(* PLC project mtcs_axes, Institute of Astronomy OntoManager 0.0.1 *)
(* stored: creationDateTime 2017-02-03T09:57:02.669561, modificationDateTime 2017-02-03T09:57:02.669561 *)

TYPE AxesIds : (AZI := 0, ABL := 1, ELE := 2, ROC := 3, RON := 4);
END_TYPE

TYPE AxesMoveUnits : (DEGREES := 0, RADIANS := 1, ARCSECONDS := 2);
END_TYPE

TYPE AxesAlphaUnits : (HOURS := 0, DEGREES := 1, RADIANS := 2);
END_TYPE

TYPE AxesDeltaUnits : (DEGREES := 0, RADIANS := 1);
END_TYPE

TYPE AxesMuUnits : (ARCSECONDS_PER_YEAR := 0, MILLIARCSECONDS_PER_YEAR := 1, DEGREES_PER_YEAR := 2, RADIANS_PER_YEAR := 3);
END_TYPE

TYPE AxesMoveVelocityUnits : (DEGREES_PER_SECOND := 0, ARCSECONDS_PER_SECOND := 1, RADIANS_PER_SECOND := 2, ARCSECONDS_PER_MINUTE := 3, ARCSECONDS_PER_HOUR := 4);
END_TYPE

TYPE AxesRotatorActivity : (NONE_ACTIVE := 0, ROC_ACTIVE := 1, RON_ACTIVE := 2);
END_TYPE

TYPE AxesParts : STRUCT
  azi : AxesAzimuthAxis;  (* The azimuth axis *)
  ele : AxesElevationAxis;  (* The elevation axis *)
  roc : AxesRotationAxis;  (* The cassegrain derotator axis *)
  ron : AxesRotationAxis;  (* The nasmyth derotator axis *)
  io : AxesIO;  (* I/O modules and drives *)
  configManager : ConfigManager;  (* The config manager (to load/save/activate configuration data) *)
  tpoint : AxesPointingModelsSetup;  (* The TPOINT models setup *)
END_STRUCT;
END_TYPE

TYPE AxesAzimuthAxisParts : STRUCT
  virtualAxis : AngularAxis;  (* The virtual AZI axis *)
  physicalAxis : AngularAxis;  (* The physical AZI axis *)
  ablAxis : AngularAxis;  (* The (anti-backlash) ABL axis *)
  lida1 : IncrementalEncoder;  (* The external (LIDA) encoder no. 1 *)
  lida2 : IncrementalEncoder;  (* The external (LIDA) encoder no. 2 *)
  lida3 : IncrementalEncoder;  (* The external (LIDA) encoder no. 3 *)
  lida4 : IncrementalEncoder;  (* The external (LIDA) encoder no. 4 *)
  absoluteEncoder : SSIEncoder;  (* The external absolute encoder *)
END_STRUCT;
END_TYPE

TYPE AxesElevationAxisParts : STRUCT
  virtualAxis : AngularAxis;  (* The virtual axis *)
  physicalAxis : AngularAxis;  (* The physical ELE axis *)
  lida1 : IncrementalEncoder;  (* The external (LIDA) encoder no. 1 *)
  lida2 : IncrementalEncoder;  (* The external (LIDA) encoder no. 2 *)
  absoluteEncoder : SSIEncoder;  (* The external absolute encoder *)
END_STRUCT;
END_TYPE

TYPE AxesRotationAxisParts : STRUCT
  virtualAxis : AngularAxis;  (* The virtual axis *)
  physicalAxis : AngularAxis;  (* The physical axis *)
END_STRUCT;
END_TYPE

TYPE AxesPointingModelSetupParts : STRUCT
  configManager : ConfigManager;  (* The config manager (to load/save/activate configuration data) *)
END_STRUCT;
END_TYPE

TYPE AxesPointingModelsSetupParts : STRUCT
  model0 : AxesPointingModelSetup;
  model1 : AxesPointingModelSetup;
  model2 : AxesPointingModelSetup;
  model3 : AxesPointingModelSetup;
  model4 : AxesPointingModelSetup;
  model5 : AxesPointingModelSetup;
  model6 : AxesPointingModelSetup;
  model7 : AxesPointingModelSetup;
  model8 : AxesPointingModelSetup;
  model9 : AxesPointingModelSetup;
END_STRUCT;
END_TYPE

TYPE AxesIOParts : STRUCT
  aziDrive : AX52XXDrive;  (* The AX5000 drive for the AZI en ROC motors *)
  ablDrive : AX52XXDrive;  (* The AX5000 drive for the ABL en RON motors *)
  eleDrive : AX52XXDrive;  (* The AX5000 drive for the ELE en FW motors *)
  TA_AZID : EtherCatDevice;  (* Telescope Axis - AZID *)
  TA_ABLD : EtherCatDevice;  (* Telescope Axis - ABLD *)
  TA_ELED : EtherCatDevice;  (* Telescope Axis - ELED *)
  TE_COU : EtherCatDevice;  (* Telescope Encoders - COU *)
  TE_EN1 : EtherCatDevice;  (* Telescope Encoders - EN1 *)
  TE_EN2 : EtherCatDevice;  (* Telescope Encoders - EN2 *)
  TE_EN3 : EtherCatDevice;  (* Telescope Encoders - EN3 *)
  TE_EN4 : EtherCatDevice;  (* Telescope Encoders - EN4 *)
  TE_EN5 : EtherCatDevice;  (* Telescope Encoders - EN5 *)
  TE_EN6 : EtherCatDevice;  (* Telescope Encoders - EN6 *)
  TE_EN7 : EtherCatDevice;  (* Telescope Encoders - EN7 *)
END_STRUCT;
END_TYPE

TYPE AxesProcesses : STRUCT
  initialize : Process;  (* Start initializing *)
  reset : Process;  (* Reset the axis (no homing) *)
  lock : Process;  (* Lock the system *)
  unlock : Process;  (* Unlock the system *)
  changeOperatingState : ChangeOperatingStateProcess;  (* Change the operating state (e.g. AUTO, MANUAL, ...) *)
  setTarget : AxesSetTargetProcess;  (* Set a new target *)
  point : AxesPointProcess;  (* Point the telescope to a new target *)
  pointRelative : AxesPointRelativeProcess;  (* Point the telescope relative to the current target *)
  stop : AxesStopProcess;  (* Stop the axes (i.e. stop pointing, tracking, moving, ...) *)
  quickStop : AxesStopProcess;  (* Quickly stop the axes (i.e. stop pointing, tracking, moving, ...) *)
  powerOn : AxesMultiPowerOnProcess;  (* Power on the axes *)
  powerOff : AxesPowerOffProcess;  (* Power off the axes *)
  doHoming : AxesDoHomingProcess;  (* Do a homing of the axes *)
  moveAbsolute : AxesMultiMoveProcess;  (* Move the axes in alt-azimuth to an absolute position *)
  moveRelative : AxesMultiMoveProcess;  (* Move the axes in alt-azimuth relative to the current position *)
  moveKnownPosition : AxesMoveKnownPositionProcess;  (* Move the axes to the given known position *)
  enablePointingModel : AxesEnablePointingModelProcess;  (* Enable a pointing model with the given name *)
  disablePointingModel : Process;  (* Disable the currently active pointing model *)
  setAlphaDeltaVelocity : AxesSetAlphaDeltaVelocityProcess;  (* Set an additional alpha/delta velocity (e.g. to track solar system objects) *)
END_STRUCT;
END_TYPE

TYPE AxesAzimuthAxisProcesses : STRUCT
  moveAbsolute : AxesMoveAbsoluteProcess;  (* Move the axis in an absolute way *)
  moveRelative : AxesMoveRelativeProcess;  (* Move the axis relative to the current position *)
  moveVelocity : AxesMoveVelocityProcess;  (* Move the axis endlessly with the given velocity *)
  reset : Process;  (* Reset the axis (no homing) *)
  moveOutOfLimitSwitch : AxesMoveOutOfLimitSwitchProcess;  (* Move out of a limit switch *)
  powerOn : AxesPowerOnProcess;  (* Power on the axis *)
  powerOff : AxesPowerOffProcess;  (* Power off the axis *)
  doHoming : AxesDoHomingProcess;  (* Do a homing of the axis *)
  stop : AxesStopProcess;  (* Stop the axis (i.e. stop pointing, tracking, moving, ...) *)
  quickStop : AxesStopProcess;  (* Quickly stop the axes (i.e. stop pointing, tracking, moving, ...) *)
  unlockBrake : AxesUnlockBrakeProcess;  (* Temporarily unlock the brake *)
  setPosition : AxesSetPositionProcess;  (* Set the axis to the given position *)
END_STRUCT;
END_TYPE

TYPE AxesElevationAxisProcesses : STRUCT
  moveAbsolute : AxesMoveAbsoluteProcess;  (* Move the axis in an absolute way *)
  moveRelative : AxesMoveRelativeProcess;  (* Move the axis relative to the current position *)
  moveVelocity : AxesMoveVelocityProcess;  (* Move the axis endlessly with the given velocity *)
  reset : Process;  (* Reset the axis (no homing) *)
  moveOutOfLimitSwitch : AxesMoveOutOfLimitSwitchProcess;  (* Move out of a limit switch *)
  powerOn : AxesPowerOnProcess;  (* Power on the axis *)
  powerOff : AxesPowerOffProcess;  (* Power off the axis *)
  doHoming : AxesDoHomingProcess;  (* Do a homing of the axis *)
  stop : AxesStopProcess;  (* Stop the axis (i.e. stop pointing, tracking, moving, ...) *)
  quickStop : AxesStopProcess;  (* Quickly stop the axes (i.e. stop pointing, tracking, moving, ...) *)
  setPosition : AxesSetPositionProcess;  (* Set the axis to the given position *)
  unlockBrake : AxesUnlockBrakeProcess;  (* Temporarily unlock the brake *)
END_STRUCT;
END_TYPE

TYPE AxesRotationAxisProcesses : STRUCT
  moveAbsolute : AxesMoveAbsoluteProcess;  (* Move the axis in an absolute way *)
  moveRelative : AxesMoveRelativeProcess;  (* Move the axis relative to the current position *)
  moveVelocity : AxesMoveVelocityProcess;  (* Move the axis endlessly with the given velocity *)
  reset : Process;  (* Reset the axis (no homing) *)
  moveOutOfLimitSwitch : AxesMoveOutOfLimitSwitchProcess;  (* Move out of a limit switch *)
  powerOn : AxesPowerOnProcess;  (* Power on the axis *)
  powerOff : AxesPowerOffProcess;  (* Power off the axis *)
  stop : AxesStopProcess;  (* Stop the axis (i.e. stop pointing, tracking, moving, ...) *)
  quickStop : AxesStopProcess;  (* Quickly stop the axes (i.e. stop pointing, tracking, moving, ...) *)
  setPosition : AxesSetPositionProcess;  (* Set the axis to the given position *)
END_STRUCT;
END_TYPE

TYPE AxesStatuses : STRUCT
  initializationStatus : InitializationStatus;
  healthStatus : HealthStatus;
  busyStatus : BusyStatus;
  operatingStatus : OperatingStatus;
  poweredStatus : PoweredStatus;
END_STRUCT;
END_TYPE

TYPE AxesTargetStatuses : STRUCT
  healthStatus : HealthStatus;
END_STRUCT;
END_TYPE

TYPE AxesFeedbackStatuses : STRUCT
  healthStatus : HealthStatus;
END_STRUCT;
END_TYPE

TYPE AxesAzimuthAxisStatuses : STRUCT
  busyStatus : BusyStatus;  (* Is the axis in a busy state? *)
  healthStatus : HealthStatus;  (* Is the axis in a healthy state? *)
  poweredStatus : PoweredStatus;  (* Is the axis powered on or off? *)
END_STRUCT;
END_TYPE

TYPE AxesElevationAxisStatuses : STRUCT
  busyStatus : BusyStatus;  (* Is the axis in a busy state? *)
  healthStatus : HealthStatus;  (* Is the axis in a healthy state? *)
  poweredStatus : PoweredStatus;  (* Is the axis powered on or off? *)
END_STRUCT;
END_TYPE

TYPE AxesRotationAxisStatuses : STRUCT
  busyStatus : BusyStatus;  (* Is the axis in a busy state? *)
  healthStatus : HealthStatus;  (* Is the axis in a healthy state? *)
  poweredStatus : PoweredStatus;  (* Is the axis powered on or off? *)
END_STRUCT;
END_TYPE

TYPE AxesPointingModelsSetupStatuses : STRUCT
  busyStatus : BusyStatus;  (* Is the pointing models setup in a busy state? *)
  healthStatus : HealthStatus;  (* Is the pointing models setup in a healthy state? *)
END_STRUCT;
END_TYPE

TYPE AxesIOStatuses : STRUCT
  healthStatus : HealthStatus;  (* Is the I/O in a healthy state? *)
END_STRUCT;
END_TYPE

TYPE AxesLocationConfig : STRUCT
  longitude : LREAL;  (* Observatory location: longitude [degrees, positive = E, negative = W] *)
  latitude : LREAL;  (* Observatory location: latitude [degrees, positive = N, negative = S] *)
  height : REAL;  (* Observatory location: height above sea-level [m] *)
  polarMotionX : REAL;  (* Earth polar motion x in degrees *)
  polarMotionY : REAL;  (* Earth polar motion y in degrees *)
  nutationDx : REAL;  (* Nutation adjustment dX in degrees *)
  nutationDy : REAL;  (* Nutation adjustment dY in degrees *)
END_STRUCT;
END_TYPE

TYPE AxesLocalConditionsConfig : STRUCT
  useTemperatureFromSensors : BOOL;  (* True if the temperature from the sensors should be used, false to use the temperature from the config *)
  configuredTemperature : REAL;  (* Local temperature in degrees, fixed by config *)
  configuredPressure : REAL;  (* Local temperature in hectoPascal = millibar, fixed by config *)
  useRelativeHumidityFromSensors : BOOL;  (* True if the temperature from the sensors should be used, false to use the temperature from the config *)
  configuredRelativeHumidity : REAL;  (* Local relative humidity as a fraction (0...1), fixed by config *)
  configuredObservingWavelength : REAL;  (* Observing wavelength in microns, fixed by config *)
  troposphericLapseRate : REAL;  (* Tropospheric lapse rate in K/m *)
END_STRUCT;
END_TYPE

TYPE AxesAzimuthConfig : STRUCT
  absoluteEncoderOffset : LREAL;  (* Offset in degrees, of the absolute encoder, w.r.t. zero *)
  absoluteEncoderInvert : BOOL;  (* TRUE to invert the counting direction of the absolute encoder *)
  lidasInvert : BOOL;  (* TRUE to invert the counting direction of the LIDAs *)
  moveOutOfLimitSwitchDistance : LREAL;  (* How many degrees should the moveOutOfLimitSwitch process try to move? *)
  positiveLimitSwitchInput : SINT;  (* Which input (0-7) represents the positive limit switch? *)
  negativeLimitSwitchInput : SINT;  (* Which input (0-7) represents the negative limit switch? *)
  minPositionLimitVirtualAxis : LREAL;  (* Limit the minimum position of the virtual axis to this value in degrees *)
  maxPositionLimitVirtualAxis : LREAL;  (* Limit the maximum position of the virtual axis to this value in degrees *)
  minPositionLimitPhysicalAxis : LREAL;  (* Limit the minimum position of the physical axis to this value in degrees *)
  maxPositionLimitPhysicalAxis : LREAL;  (* Limit the maximum position of the physical axis to this value in degrees *)
  velocityLimit : LREAL;  (* Limit the velocity of the axis to this value in degrees/sec *)
  accelerationLimit : LREAL;  (* Limit the acceleration (or deceleration) of the axis to this value in degrees/sec^2 *)
  minPositionSetpoint : LREAL;  (* The minimum position setpoint of the axis in degrees (should be a bit before the minPositionLimit) *)
  maxPositionSetpoint : LREAL;  (* The maximum position setpoint of the axis in degrees (should be a bit before the maxPositionLimit) *)
  maxVelocitySetpoint : LREAL;  (* The maximum velocity setpoint of the axis in degrees/sec *)
  maxAccelerationSetpoint : LREAL;  (* The maximum acceleration setpoint of the axis in degrees/sec^2 *)
  slipLimit : LREAL;  (* If the difference between the LIDA-encoder and motor-encoder positions is above this value in degrees, then we have detected slip *)
  ablMaxTorqueRiseSpeed : LREAL;  (* The ABL torque can rise maximum ... Nm/s on the telescope axis (always >0) *)
  ablMaxTorqueFallSpeed : LREAL;  (* The ABL torque can fall maximum ... Nm/s on the telescope axis (always >0) *)
  ablMaxTorque : LREAL;  (* The maximum ABL torque in Nm/s on the telescope axis (always >0) *)
  ablMinTorque : LREAL;  (* The minimum ABL torque in Nm/s on the telescope axis (always >0) *)
  ablZeroAccTorque : LREAL;  (* The ABL torque when the axis is not accelerating or decelerating (always >0) *)
  ablTorqueOutputOverride : LREAL;  (* Scale the ABL output torque by this fraction value (only for testing purposes, must be 1 normally!) *)
  ablPositiveTorque : BOOL;  (* True if a positive torque must be applied, false if a negative torque must be applied *)
  aziAndAblSameDirection : BOOL;  (* True if the AZI and ABL axes rotate in the same direction? *)
  homingHomePosition : LREAL;  (* The position of the homing mark (in degrees), with respect to the absolute zero *)
  homingStartAbsEncPosition : LREAL;  (* Absolute encoder position where the homing should go to first, in degrees *)
  homingGotoStartVelocity : LREAL;  (* Velocity when going to the start position, in degrees/sec *)
  homingVelocity : LREAL;  (* Velocity to search for the homing mark, in degrees/sec *)
  homingRange : LREAL;  (* Maximum distance to be covered while searching for the homing mark, in degrees *)
  quickStopDeceleration : LREAL;  (* Quick stop deceleration, in degrees/sec2 *)
  quickStopJerk : LREAL;  (* Quick stop jerk, in degrees/sec3 *)
END_STRUCT;
END_TYPE

TYPE AxesElevationConfig : STRUCT
  absoluteEncoderOffset : LREAL;  (* Offset in degrees, of the absolute encoder, w.r.t. zero *)
  absoluteEncoderInvert : BOOL;  (* TRUE to invert the counting direction *)
  lidasInvert : BOOL;  (* TRUE to invert the counting direction of the LIDAs *)
  moveOutOfLimitSwitchDistance : LREAL;  (* How many degrees should the moveOutOfLimitSwitch process try to move? *)
  positiveLimitSwitchInput : SINT;  (* Which input (0-7) represents the positive limit switch? *)
  negativeLimitSwitchInput : SINT;  (* Which input (0-7) represents the negative limit switch? *)
  minPositionLimitVirtualAxis : LREAL;  (* Limit the minimum position of the axis to this value in degrees, of the virtual axis *)
  maxPositionLimitVirtualAxis : LREAL;  (* Limit the maximum position of the axis to this value in degrees, of the virtual axis *)
  minPositionLimitPhysicalAxis : LREAL;  (* Limit the minimum position of the axis to this value in degrees, of the physical axis *)
  maxPositionLimitPhysicalAxis : LREAL;  (* Limit the maximum position of the axis to this value in degrees, of the physical axis *)
  velocityLimit : LREAL;  (* Limit the velocity of the axis to this value in degrees/sec *)
  accelerationLimit : LREAL;  (* Limit the acceleration (or deceleration) of the axis to this value in degrees/sec^2 *)
  minPositionSetpoint : LREAL;  (* The minimum position setpoint of the axis in degrees *)
  maxPositionSetpoint : LREAL;  (* The maximum position setpoint of the axis in degrees *)
  maxVelocitySetpoint : LREAL;  (* The maximum velocity setpoint of the axis in degrees/sec *)
  maxAccelerationSetpoint : LREAL;  (* The maximum acceleration setpoint of the axis in degrees/sec^2 *)
  slipLimit : LREAL;  (* If the difference between the LIDA-encoder and motor-encoder positions is above this value in degrees, then we have detected slip *)
  homingHomePosition : LREAL;  (* The position of the homing mark (in degrees), with respect to the absolute zero *)
  homingStartAbsEncPosition : LREAL;  (* Absolute encoder position where the homing should go to first, in degrees *)
  homingGotoStartVelocity : LREAL;  (* Velocity when going to the start position, in degrees/sec *)
  homingVelocity : LREAL;  (* Velocity to search for the homing mark, in degrees/sec *)
  homingRange : LREAL;  (* Maximum distance to be covered while searching for the homing mark, in degrees *)
  quickStopDeceleration : LREAL;  (* Quick stop deceleration, in degrees/sec2 *)
  quickStopJerk : LREAL;  (* Quick stop jerk, in degrees/sec3 *)
END_STRUCT;
END_TYPE

TYPE AxesRotationConfig : STRUCT
  motorEncoderOffset : LREAL;  (* Offset in degrees, of the absolute motor encoder, w.r.t. zero *)
  moveOutOfLimitSwitchDistance : LREAL;  (* How many degrees should the moveOutOfLimitSwitch process try to move? *)
  positiveLimitSwitchInput : SINT;  (* Which input (0-7) represents the positive limit switch? *)
  negativeLimitSwitchInput : SINT;  (* Which input (0-7) represents the negative limit switch? *)
  minPositionLimitVirtualAxis : LREAL;  (* Limit the minimum position of the axis to this value in degrees, of the virtual axis *)
  maxPositionLimitVirtualAxis : LREAL;  (* Limit the maximum position of the axis to this value in degrees, of the virtual axis *)
  minPositionLimitPhysicalAxis : LREAL;  (* Limit the minimum position of the axis to this value in degrees, of the physical axis *)
  maxPositionLimitPhysicalAxis : LREAL;  (* Limit the maximum position of the axis to this value in degrees, of the physical axis *)
  velocityLimit : LREAL;  (* Limit the velocity of the axis to this value in degrees/sec *)
  accelerationLimit : LREAL;  (* Limit the acceleration (or deceleration) of the axis to this value in degrees/sec^2 *)
  minPositionSetpoint : LREAL;  (* The minimum position setpoint of the axis in degrees *)
  maxPositionSetpoint : LREAL;  (* The maximum position setpoint of the axis in degrees *)
  maxVelocitySetpoint : LREAL;  (* The maximum velocity setpoint of the axis in degrees/sec *)
  maxAccelerationSetpoint : LREAL;  (* The maximum acceleration setpoint of the axis in degrees/sec^2 *)
  quickStopDeceleration : LREAL;  (* Quick stop deceleration, in degrees/sec2 *)
  quickStopJerk : LREAL;  (* Quick stop jerk, in degrees/sec3 *)
END_STRUCT;
END_TYPE

TYPE AxesKnownPositionConfig : STRUCT
  name : STRING;  (* The name of the position (e.g. 'PARK') *)
  allowObserver : BOOL;  (* Can an observer switch to this position? *)
  azi : LREAL;  (* Azimuth in degrees *)
  ele : LREAL;  (* Elevation in degrees *)
  roc : LREAL;  (* Cassegrain rotation in degrees *)
  ron : LREAL;  (* Nasmyth B rotation in degrees *)
  doAzi : BOOL;  (* Change the azimuth axis to the 'azi' position *)
  doEle : BOOL;  (* Change the elevation axis to the 'ele' position *)
  doRoc : BOOL;  (* Change the cassegrain rotation axis to the 'roc' position *)
  doRon : BOOL;  (* Change the nasmyth rotation axis to the 'ron' position *)
END_STRUCT;
END_TYPE

TYPE AxesKnownPositionsConfig : STRUCT
  position0 : AxesKnownPositionConfig;  (* Known position 0 *)
  position1 : AxesKnownPositionConfig;  (* Known position 1 *)
  position2 : AxesKnownPositionConfig;  (* Known position 2 *)
  position3 : AxesKnownPositionConfig;  (* Known position 3 *)
  position4 : AxesKnownPositionConfig;  (* Known position 4 *)
  position5 : AxesKnownPositionConfig;  (* Known position 5 *)
  position6 : AxesKnownPositionConfig;  (* Known position 6 *)
  position7 : AxesKnownPositionConfig;  (* Known position 7 *)
  position8 : AxesKnownPositionConfig;  (* Known position 8 *)
  position9 : AxesKnownPositionConfig;  (* Known position 9 *)
  position10 : AxesKnownPositionConfig;  (* Known position 10 *)
  position11 : AxesKnownPositionConfig;  (* Known position 11 *)
  position12 : AxesKnownPositionConfig;  (* Known position 12 *)
  position13 : AxesKnownPositionConfig;  (* Known position 13 *)
  position14 : AxesKnownPositionConfig;  (* Known position 14 *)
  position15 : AxesKnownPositionConfig;  (* Known position 15 *)
  position16 : AxesKnownPositionConfig;  (* Known position 16 *)
  position17 : AxesKnownPositionConfig;  (* Known position 17 *)
  position18 : AxesKnownPositionConfig;  (* Known position 18 *)
  position19 : AxesKnownPositionConfig;  (* Known position 19 *)
END_STRUCT;
END_TYPE

TYPE AxesConfig : STRUCT
  location : AxesLocationConfig;  (* Location of the observatory *)
  localConditions : AxesLocalConditionsConfig;  (* Location of the observatory *)
  knownPositions : AxesKnownPositionsConfig;  (* Known (predefined) positions (e.g. could be Park, Cover, Park winter, Mirror washing, ...) *)
  azi : AxesAzimuthConfig;  (* Azimuth axis *)
  ele : AxesElevationConfig;  (* Elevation axis *)
  roc : AxesRotationConfig;  (* Cassegrain rotation axis *)
  ron : AxesRotationConfig;  (* Nasmyth rotation axis *)
  cassegrainRotatorName : STRING;  (* Name of the Cassegrain rotator *)
  nasmythRotatorName : STRING;  (* Name of the Nasmyth rotator *)
  rocGuiAngle : LREAL;  (* Amgle to show ROC in the GUI *)
  ronGuiAngle : LREAL;  (* Amgle to show RON in the GUI *)
  knownPositionToleranceAzi : LREAL;  (* Tolerance (in degrees) to determine if the telescope is at a known position in azi direction *)
  knownPositionToleranceEle : LREAL;  (* Tolerance (in degrees) to determine if the telescope is at a known position in ele direction *)
  knownPositionToleranceRoc : LREAL;  (* Tolerance (in degrees) to determine if the telescope is at a known position in roc direction *)
  knownPositionToleranceRon : LREAL;  (* Tolerance (in degrees) to determine if the telescope is at a known position in ron direction *)
  rocPositionAngleSign : INT;  (* -1 to invert the sign of the PA for the cas derotator, 1 for positive *)
  ronPositionAngleSign : INT;  (* -1 to invert the sign of the PA for the cas derotator, 1 for positive *)
  tpointAziSign : INT;  (* -1 or 1 to invert input for TPOINT: A *)
  tpointEleSign : INT;  (* -1 or 1 to invert input for TPOINT: E *)
  tpointDeltaAziSign : INT;  (* -1 or 1 to invert input for TPOINT: DA *)
  tpointDeltaEleSign : INT;  (* -1 or 1 to invert input for TPOINT: DE *)
  tpointOldFormulas : BOOL;  (* True to use the old formulas *)
  tpointConvertRawAlphaDelta : BOOL;  (* If True, raw encoder values will be converted to feedback.alpha and feedback.delta, instead of corrected encoder values. Only use for tech stuff! *)
END_STRUCT;
END_TYPE

TYPE AxesPointingModelConfig : STRUCT
  name : STRING;  (* This name can be matched against the instrument name in the MTCS config and the focal station name in the M3 config. *)
  IE : LREAL;  (* Index error in elevation *)
  IA : LREAL;  (* Index error in azimuth *)
  CA : LREAL;  (* Nonperpendicularity of elevation and pointing axes *)
  AN : LREAL;  (* NS misalignment of azimuth axis *)
  AW : LREAL;  (* EW misalignment of azimuth axis *)
  NPAE : LREAL;  (* Nonperpendicularity of azimuth and elevation axes *)
  NRX : LREAL;  (* Horizontal displacement of Nasmyth rotation *)
  NRY : LREAL;  (* Vertical displacement of Nasmyth rotation *)
  ACES : LREAL;  (* Az centering error (sin component) *)
  ACEC : LREAL;  (* Az centering error (cos component) *)
  ECES : LREAL;  (* El centering error (sin component) *)
  ECEC : LREAL;  (* El centering error (cos component) *)
  TF : LREAL;  (* Tube flexure - sin(zeta) law *)
  TX : LREAL;  (* Tube flexure - tan(zeta) law *)
  FLOP : LREAL;  (* Constant vertical displacement *)
  POX : LREAL;  (* The x-coordinate of a pointing origin on a derotator *)
  POY : LREAL;  (* The y-coordinate of a pointing origin on a derotator *)
END_STRUCT;
END_TYPE

TYPE AxesSetTargetProcessArgs : STRUCT
  alphaUnits : AxesAlphaUnits;  (* The units in which alpha is given *)
  alpha : LREAL;  (* Right ascention, in the units of the alphaUnits argument *)
  deltaUnits : AxesDeltaUnits;  (* The units in which delta is given *)
  delta : LREAL;  (* Declination, in the units of the deltaUnits argument *)
  muUnits : AxesMuUnits;  (* The units in which muAlpha and muDelta are given *)
  muAlpha : LREAL;  (* Right ascention proper motion, the units of muUmits (do not multiply by cos(delta)!) *)
  muDelta : LREAL;  (* Declination proper motion, in radians/year *)
  parallax : LREAL;  (* Object parallax, in arcseconds *)
  radialVelocity : LREAL;  (* Object radial velocity, in km/s *)
  epoch : LREAL := 2000;  (* Epoch, e.g. 2000.0 *)
END_STRUCT;
END_TYPE

TYPE AxesPointProcessArgs : STRUCT
  alphaUnits : AxesAlphaUnits;  (* The units in which alpha is given *)
  alpha : LREAL;  (* Right ascention, in the units of the alphaUnits argument *)
  deltaUnits : AxesDeltaUnits;  (* The units in which delta is given *)
  delta : LREAL;  (* Declination, in the units of the deltaUnits argument *)
  muUnits : AxesMuUnits;  (* The units in which muAlpha and muDelta are given *)
  muAlpha : LREAL;  (* Right ascention proper motion, the units of muUmits (do not multiply by cos(delta)!) *)
  muDelta : LREAL;  (* Declination proper motion, in radians/year *)
  parallax : LREAL;  (* Object parallax, in arcseconds *)
  radialVelocity : LREAL;  (* Object radial velocity, in km/s *)
  epoch : LREAL := 2000;  (* Epoch, e.g. 2000.0 *)
  tracking : BOOL := TRUE;  (* True to start tracking the object, false to Only do a pointing *)
  rotUnits : AxesMoveUnits;  (* Units of the 'rot', 'roc' and 'ron' arguments (RADIANS, DEGREES, ARCSECONDS, ...) *)
  rotOffset : LREAL;  (* Offset to move the currently active rotator (incompatible with 'roc' and 'ron' args) *)
  rocOffset : LREAL;  (* Offset to move the cassegrain rotation axis (incompatible with 'rot' arg) *)
  ronOffset : LREAL;  (* Offset to move the nasmyth rotation axis (incompatible with 'rot' arg) *)
  doRotOffset : BOOL;  (* True to move the currently active rotator, false to leave it untouched *)
  doRocOffset : BOOL;  (* True to move the cassegrain rotation axis, false to leave it untouched *)
  doRonOffset : BOOL;  (* True to move the nasmyth rotation axis, false to leave it untouched *)
END_STRUCT;
END_TYPE

TYPE AxesPointRelativeProcessArgs : STRUCT
  alphaUnits : AxesAlphaUnits;  (* The units in which alpha is given *)
  alpha : LREAL;  (* Right ascention, in the units of the alphaUnits argument *)
  deltaUnits : AxesDeltaUnits;  (* The units in which delta is given *)
  delta : LREAL;  (* Declination, in the units of the deltaUnits argument *)
END_STRUCT;
END_TYPE

TYPE AxesMoveRelativeProcessArgs : STRUCT
  units : AxesMoveUnits;  (* Units of the 'value' argument (RADIANS, DEGREES, ARCSECONDS, ...) *)
  value : LREAL;  (* Move the axis with this value (which units depends on the 'units' argument) *)
END_STRUCT;
END_TYPE

TYPE AxesMoveAbsoluteProcessArgs : STRUCT
  units : AxesMoveUnits;  (* Units of the 'value' argument (RADIANS, DEGREES, ARCSECONDS, ...) *)
  value : LREAL;  (* Move the axis to this value (which units depends on the 'units' argument) + the optional offset *)
  offset : LREAL;  (* Optional extra offset (which will not be added to the 'startPos' *)
END_STRUCT;
END_TYPE

TYPE AxesMoveKnownPositionProcessArgs : STRUCT
  name : STRING;  (* Name of the position to move to *)
END_STRUCT;
END_TYPE

TYPE AxesMoveVelocityProcessArgs : STRUCT
  units : AxesMoveVelocityUnits;  (* Units of the 'value' argument (RADIANS_PER_SECOND, DEGREES_PER_SECOND, ...) *)
  value : LREAL;  (* Move the axis with this velocity (which units depends on the 'units' argument) *)
END_STRUCT;
END_TYPE

TYPE AxesMoveOutOfLimitSwitchProcessArgs : STRUCT
  switch : LimitSwitches;  (* Positive or negative limit switch *)
END_STRUCT;
END_TYPE

TYPE AxesMultiPowerOnProcessArgs : STRUCT
  azi : BOOL;  (* TRUE to power on AZI *)
  ele : BOOL;  (* TRUE to power on ELE *)
  roc : BOOL;  (* TRUE to power on ROC *)
  ron : BOOL;  (* TRUE to power on RON *)
  fw : BOOL;  (* TRUE to power on FW *)
END_STRUCT;
END_TYPE

TYPE AxesSetAlphaDeltaVelocityProcessArgs : STRUCT
  units : AxesMoveVelocityUnits;  (* Units of the alphaVelocity and deltaVelocity *)
  alphaVelocity : LREAL;  (* Velocity in alpha direction *)
  deltaVelocity : LREAL;  (* Velocity in delta direction *)
END_STRUCT;
END_TYPE

TYPE AxesMultiMoveProcessArgs : STRUCT
  units : AxesMoveUnits;  (* Units of the 'azi', 'ele', 'roc' and 'ron' arguments (RADIANS, DEGREES, ARCSECONDS, ...) *)
  azi : LREAL;  (* Angle to move the azimuth axis *)
  ele : LREAL;  (* Angle to move the elevation axis *)
  rot : LREAL;  (* Angle to move the currently active rotator (incompatible with 'roc' and 'ron' args) *)
  roc : LREAL;  (* Angle to move the cassegrain rotation axis (incompatible with 'rot' arg) *)
  ron : LREAL;  (* Angle to move the nasmyth rotation axis (incompatible with 'rot' arg) *)
  doAzi : BOOL;  (* True to move the azimuth axis, false to leave it untouched *)
  doEle : BOOL;  (* True to move the elevation axis, false to leave it untouched *)
  doRot : BOOL;  (* True to move the currently active rotator, false to leave it untouched *)
  doRoc : BOOL;  (* True to move the cassegrain rotation axis, false to leave it untouched *)
  doRon : BOOL;  (* True to move the nasmyth rotation axis, false to leave it untouched *)
  preferMostTravel : BOOL := FALSE;  (* Only in case of relative movement during tracking: If possible, go to the position where there is most travel (if the telescope is tracking). If false, it will go there the quickest way possible. *)
END_STRUCT;
END_TYPE

TYPE AxesEnablePointingModelProcessArgs : STRUCT
  name : STRING;  (* Name of the pointing model *)
END_STRUCT;
END_TYPE

TYPE AxesUnlockBrakeProcessArgs : STRUCT
  seconds : LREAL := 10.0;  (* Unlock the brake for this number of seconds (0 means forever) *)
END_STRUCT;
END_TYPE

TYPE AxesSetPositionProcessArgs : STRUCT
  value : LREAL;  (* New position to be taken over by the axis *)
END_STRUCT;
END_TYPE

FUNCTION_BLOCK SM_Axes
  VAR_INPUT
    {attribute 'OPC.UA.DA' := '1'}
    {attribute 'OPC.UA.DA.Access' := '1'}
    editableConfig : AxesConfig;  (* Editable configuration of the Axes subsystem *)
    {attribute 'OPC.UA.DA' := '1'}
    {attribute 'OPC.UA.DA.Access' := '1'}
    fromCppAxes AT %I* : TmcToPlcAxes;  (* Data from the C++ task *)
  END_VAR
  VAR_OUTPUT
    {attribute 'OPC.UA.DA' := '1'}
    {attribute 'OPC.UA.DA.Access' := '1'}
    actualStatus : STRING;  (* Current status description *)
    previousStatus : STRING;  (* Previous status description *)
    {attribute 'OPC.UA.DA' := '1'}
    {attribute 'OPC.UA.DA.Access' := '1'}
    isPoweredOffByPersonInDome : BOOL;  (* True if the axes are powered off due to a person entering the dome *)
    {attribute 'OPC.UA.DA' := '1'}
    {attribute 'OPC.UA.DA.Access' := '1'}
    isPointing : BOOL;  (* True if the telescope is pointing *)
    {attribute 'OPC.UA.DA' := '1'}
    {attribute 'OPC.UA.DA.Access' := '1'}
    isLimitsReached : BOOL;  (* True if a positiom limit is reached *)
    {attribute 'OPC.UA.DA' := '1'}
    {attribute 'OPC.UA.DA.Access' := '1'}
    isTracking : BOOL;  (* True if the telescope is tracking *)
    {attribute 'OPC.UA.DA' := '1'}
    {attribute 'OPC.UA.DA.Access' := '1'}
    isOffsetting : BOOL;  (* True if the telescope is offsetting (movin *)
    {attribute 'OPC.UA.DA' := '1'}
    {attribute 'OPC.UA.DA.Access' := '1'}
    isAtKnownPosition : BOOL;  (* True if the telescope is at a known position *)
    {attribute 'OPC.UA.DA' := '1'}
    {attribute 'OPC.UA.DA.Access' := '1'}
    isPointingModelActive : BOOL;  (* Is a pointing model currently active? *)
    {attribute 'OPC.UA.DA' := '1'}
    {attribute 'OPC.UA.DA.Access' := '1'}
    activeRotator : AxesRotatorActivity;  (* Which rotator is active? *)
    {attribute 'OPC.UA.DA' := '1'}
    {attribute 'OPC.UA.DA.Access' := '1'}
    actualKnownPositionName : STRING;  (* Name of the known position if isAtKnownPosition is True *)
    {attribute 'OPC.UA.DA' := '1'}
    {attribute 'OPC.UA.DA.Access' := '1'}
    config : AxesConfig;  (* Active configuration of the Axes subsystem *)
    {attribute 'OPC.UA.DA' := '1'}
    {attribute 'OPC.UA.DA.Access' := '1'}
    toCppAxes AT %Q* : TmcFromPlcAxes;  (* Data to the C++ task *)
    {attribute 'OPC.UA.DA' := '1'}
    {attribute 'OPC.UA.DA.Access' := '1'}
    activePointingModel : AxesPointingModelConfig;  (* Currently active TPoint model (if isPointingModelActive is TRUE) *)
    {attribute 'OPC.UA.DA' := '1'}
    {attribute 'OPC.UA.DA.Access' := '1'}
    activePointingModelNumber : INT;  (* Number of the currently active TPoint model (if isPointingModelActive is TRUE), -1 if no model is active *)
    {attribute 'OPC.UA.DA' := '1'}
    {attribute 'OPC.UA.DA.Access' := '1'}
    target : AxesTarget;  (* The actual target *)
    {attribute 'OPC.UA.DA' := '1'}
    {attribute 'OPC.UA.DA.Access' := '1'}
    feedback : AxesFeedback;  (* The actual feedback *)
    statuses : AxesStatuses;  (* Statuses of the state machine *)
    parts : AxesParts;  (* Parts of the state machine *)
    processes : AxesProcesses;  (* Processes of the state machine *)
  END_VAR
  VAR_IN_OUT
    {attribute 'OPC.UA.DA' := '0'}
    timing : ServicesTiming;  (* Reference to the timing service *)
    {attribute 'OPC.UA.DA' := '0'}
    motionBlocking : SafetyMotionBlocking;  (* Reference to the motion blocking safety *)
    {attribute 'OPC.UA.DA' := '0'}
    domeAccess : SafetyDomeAccess;  (* Reference to the dome access safety *)
    {attribute 'OPC.UA.DA' := '0'}
    operatorStatus : OperatorStatus;  (* Shared operator status *)
    {attribute 'OPC.UA.DA' := '0'}
    activityStatus : ActivityStatus;  (* Shared activity status *)
    {attribute 'OPC.UA.DA' := '0'}
    activeInstrument : InstrumentConfig;  (* Instrument config *if* isInstrumentActive is TRUE *)
    {attribute 'OPC.UA.DA' := '0'}
    isInstrumentActive : BOOL;  (* Is an instrument currently active (i.e. is M3 static at a known position?) *)
  END_VAR

            parts.azi(
    isEnabled := operatorStatus.tech,
    id := AxesIds.AZI,
    config := config.azi,
    aziDriveChannel := parts.io.parts.aziDrive.parts.channelA,
    ablDriveChannel := parts.io.parts.ablDrive.parts.channelA,
    aziMainDriveChannel := parts.io.parts.aziDrive.parts.channelA,
    ablMainDriveChannel := parts.io.parts.ablDrive.parts.channelA);
parts.ele(
    isEnabled := operatorStatus.tech,
    id := AxesIds.ELE,
    config := config.ele,
    driveChannel := parts.io.parts.eleDrive.parts.channelA,
    mainDriveChannel := parts.io.parts.eleDrive.parts.channelA);
parts.roc(
    isEnabled := operatorStatus.tech,
    id := AxesIds.ROC,
    config := config.roc,
    driveChannel := parts.io.parts.aziDrive.parts.channelB,
    mainDriveChannel := parts.io.parts.aziDrive.parts.channelA);
parts.ron(
    isEnabled := operatorStatus.tech,
    id := AxesIds.RON,
    config := config.ron,
    driveChannel := parts.io.parts.ablDrive.parts.channelB,
    mainDriveChannel := parts.io.parts.ablDrive.parts.channelA);
parts.io( isEnabled := operatorStatus.tech );
parts.configManager( isEnabled := operatorStatus.tech );
parts.tpoint( isEnabled := operatorStatus.tech );
statuses.initializationStatus();
statuses.healthStatus(
    isGood := feedback.statuses.healthStatus.isGood AND (target.statuses.healthStatus.isGood AND (parts.azi.statuses.healthStatus.isGood AND (parts.ele.statuses.healthStatus.isGood AND (parts.roc.statuses.healthStatus.isGood AND (parts.ron.statuses.healthStatus.isGood AND (parts.configManager.statuses.healthStatus.isGood AND (parts.tpoint.statuses.healthStatus.isGood AND (parts.io.statuses.healthStatus.isGood AND (processes.initialize.statuses.healthStatus.isGood AND (processes.reset.statuses.healthStatus.isGood AND (processes.lock.statuses.healthStatus.isGood AND (processes.unlock.statuses.healthStatus.isGood AND (processes.changeOperatingState.statuses.healthStatus.isGood AND (processes.setTarget.statuses.healthStatus.isGood AND (processes.point.statuses.healthStatus.isGood AND (processes.pointRelative.statuses.healthStatus.isGood AND (processes.stop.statuses.healthStatus.isGood AND (processes.quickStop.statuses.healthStatus.isGood AND (processes.powerOn.statuses.healthStatus.isGood AND (processes.powerOff.statuses.healthStatus.isGood AND (processes.doHoming.statuses.healthStatus.isGood AND (processes.moveAbsolute.statuses.healthStatus.isGood AND (processes.moveRelative.statuses.healthStatus.isGood AND (processes.moveKnownPosition.statuses.healthStatus.isGood AND (processes.enablePointingModel.statuses.healthStatus.isGood AND (processes.disablePointingModel.statuses.healthStatus.isGood AND processes.setAlphaDeltaVelocity.statuses.healthStatus.isGood)))))))))))))))))))))))))),
    hasWarning := feedback.statuses.healthStatus.hasWarning OR (target.statuses.healthStatus.hasWarning OR (parts.azi.statuses.healthStatus.hasWarning OR (parts.ele.statuses.healthStatus.hasWarning OR (parts.roc.statuses.healthStatus.hasWarning OR (parts.ron.statuses.healthStatus.hasWarning OR (parts.configManager.statuses.healthStatus.hasWarning OR (parts.tpoint.statuses.healthStatus.hasWarning OR (parts.io.statuses.healthStatus.hasWarning OR (processes.initialize.statuses.healthStatus.hasWarning OR (processes.reset.statuses.healthStatus.hasWarning OR (processes.lock.statuses.healthStatus.hasWarning OR (processes.unlock.statuses.healthStatus.hasWarning OR (processes.changeOperatingState.statuses.healthStatus.hasWarning OR (processes.setTarget.statuses.healthStatus.hasWarning OR (processes.point.statuses.healthStatus.hasWarning OR (processes.pointRelative.statuses.healthStatus.hasWarning OR (processes.stop.statuses.healthStatus.hasWarning OR (processes.quickStop.statuses.healthStatus.hasWarning OR (processes.powerOn.statuses.healthStatus.hasWarning OR (processes.powerOff.statuses.healthStatus.hasWarning OR (processes.doHoming.statuses.healthStatus.hasWarning OR (processes.moveAbsolute.statuses.healthStatus.hasWarning OR (processes.moveRelative.statuses.healthStatus.hasWarning OR (processes.moveKnownPosition.statuses.healthStatus.hasWarning OR (processes.enablePointingModel.statuses.healthStatus.hasWarning OR (processes.disablePointingModel.statuses.healthStatus.hasWarning OR processes.setAlphaDeltaVelocity.statuses.healthStatus.hasWarning)))))))))))))))))))))))))));
statuses.busyStatus( isBusy := parts.azi.statuses.busyStatus.busy OR (parts.ele.statuses.busyStatus.busy OR (parts.roc.statuses.busyStatus.busy OR (parts.ron.statuses.busyStatus.busy OR (parts.configManager.statuses.busyStatus.busy OR (parts.tpoint.statuses.busyStatus.busy OR (processes.initialize.statuses.busyStatus.busy OR (processes.reset.statuses.busyStatus.busy OR (processes.lock.statuses.busyStatus.busy OR (processes.unlock.statuses.busyStatus.busy OR (processes.changeOperatingState.statuses.busyStatus.busy OR (processes.setTarget.statuses.busyStatus.busy OR (processes.point.statuses.busyStatus.busy OR (processes.pointRelative.statuses.busyStatus.busy OR (processes.stop.statuses.busyStatus.busy OR (processes.quickStop.statuses.busyStatus.busy OR (processes.powerOn.statuses.busyStatus.busy OR (processes.powerOff.statuses.busyStatus.busy OR (processes.doHoming.statuses.busyStatus.busy OR (processes.moveAbsolute.statuses.busyStatus.busy OR (processes.moveRelative.statuses.busyStatus.busy OR (processes.moveKnownPosition.statuses.busyStatus.busy OR (processes.enablePointingModel.statuses.busyStatus.busy OR (processes.disablePointingModel.statuses.busyStatus.busy OR processes.setAlphaDeltaVelocity.statuses.busyStatus.busy))))))))))))))))))))))) );
statuses.operatingStatus( superState := statuses.initializationStatus.initialized );
statuses.poweredStatus();
processes.initialize( isEnabled := statuses.initializationStatus.shutdown OR (statuses.initializationStatus.initializingFailed OR statuses.initializationStatus.initialized) );
processes.reset( isEnabled := TRUE );
processes.lock( isEnabled := operatorStatus.tech AND statuses.initializationStatus.initialized );
processes.unlock( isEnabled := operatorStatus.tech AND statuses.initializationStatus.locked );
processes.changeOperatingState( isEnabled := statuses.busyStatus.idle AND (statuses.initializationStatus.initialized AND operatorStatus.tech) );
processes.setTarget( isEnabled := statuses.initializationStatus.initialized AND operatorStatus.tech );
processes.point( isEnabled := statuses.initializationStatus.initialized AND (statuses.busyStatus.idle AND statuses.poweredStatus.enabled) );
processes.pointRelative( isEnabled := statuses.initializationStatus.initialized AND (statuses.busyStatus.idle AND statuses.poweredStatus.enabled) );
processes.stop( isEnabled := statuses.initializationStatus.initialized );
processes.quickStop( isEnabled := statuses.initializationStatus.initialized );
processes.powerOn( isEnabled := statuses.initializationStatus.initialized AND processes.powerOn.statuses.busyStatus.idle );
processes.powerOff( isEnabled := statuses.initializationStatus.initialized AND processes.powerOff.statuses.busyStatus.idle );
processes.doHoming( isEnabled := operatorStatus.tech );
processes.moveAbsolute( isEnabled := statuses.initializationStatus.initialized AND (statuses.busyStatus.idle AND statuses.poweredStatus.enabled) );
processes.moveRelative( isEnabled := statuses.initializationStatus.initialized AND (statuses.busyStatus.idle AND statuses.poweredStatus.enabled) );
processes.moveKnownPosition( isEnabled := statuses.initializationStatus.initialized AND (statuses.busyStatus.idle AND statuses.poweredStatus.enabled) );
processes.enablePointingModel( isEnabled := statuses.busyStatus.idle );
processes.disablePointingModel( isEnabled := statuses.busyStatus.idle );
processes.setAlphaDeltaVelocity( isEnabled := statuses.initializationStatus.initialized AND statuses.busyStatus.idle );

          

{attribute 'TcRpcEnable' := '1'}
METHOD initialize : RequestResults
                  initialize := THIS^.processes.initialize.request();

                
END_METHOD

{attribute 'TcRpcEnable' := '1'}
METHOD reset : RequestResults
                  reset := THIS^.processes.reset.request();

                
END_METHOD

{attribute 'TcRpcEnable' := '1'}
METHOD lock : RequestResults
                  lock := THIS^.processes.lock.request();

                
END_METHOD

{attribute 'TcRpcEnable' := '1'}
METHOD unlock : RequestResults
                  unlock := THIS^.processes.unlock.request();

                
END_METHOD

{attribute 'TcRpcEnable' := '1'}
METHOD changeOperatingState : RequestResults
  VAR_INPUT
    state : OperatingStates;
  END_VAR
                  changeOperatingState := THIS^.processes.changeOperatingState.request( state := state );

                
END_METHOD

{attribute 'TcRpcEnable' := '1'}
METHOD setTarget : RequestResults
  VAR_INPUT
    alphaUnits : AxesAlphaUnits;
    alpha : LREAL;
    deltaUnits : AxesDeltaUnits;
    delta : LREAL;
    muUnits : AxesMuUnits;
    muAlpha : LREAL;
    muDelta : LREAL;
    parallax : LREAL;
    radialVelocity : LREAL;
    epoch : LREAL;
  END_VAR
                  setTarget := THIS^.processes.setTarget.request(
    alphaUnits := alphaUnits,
    alpha := alpha,
    deltaUnits := deltaUnits,
    delta := delta,
    muUnits := muUnits,
    muAlpha := muAlpha,
    muDelta := muDelta,
    parallax := parallax,
    radialVelocity := radialVelocity,
    epoch := epoch);

                
END_METHOD

{attribute 'TcRpcEnable' := '1'}
METHOD point : RequestResults
  VAR_INPUT
    alphaUnits : AxesAlphaUnits;
    alpha : LREAL;
    deltaUnits : AxesDeltaUnits;
    delta : LREAL;
    muUnits : AxesMuUnits;
    muAlpha : LREAL;
    muDelta : LREAL;
    parallax : LREAL;
    radialVelocity : LREAL;
    epoch : LREAL;
    tracking : BOOL;
    rotUnits : AxesMoveUnits;
    rotOffset : LREAL;
    rocOffset : LREAL;
    ronOffset : LREAL;
    doRotOffset : BOOL;
    doRocOffset : BOOL;
    doRonOffset : BOOL;
  END_VAR
                  point := THIS^.processes.point.request(
    alphaUnits := alphaUnits,
    alpha := alpha,
    deltaUnits := deltaUnits,
    delta := delta,
    muUnits := muUnits,
    muAlpha := muAlpha,
    muDelta := muDelta,
    parallax := parallax,
    radialVelocity := radialVelocity,
    epoch := epoch,
    tracking := tracking,
    rotUnits := rotUnits,
    rotOffset := rotOffset,
    rocOffset := rocOffset,
    ronOffset := ronOffset,
    doRotOffset := doRotOffset,
    doRocOffset := doRocOffset,
    doRonOffset := doRonOffset);

                
END_METHOD

{attribute 'TcRpcEnable' := '1'}
METHOD pointRelative : RequestResults
  VAR_INPUT
    alphaUnits : AxesAlphaUnits;
    alpha : LREAL;
    deltaUnits : AxesDeltaUnits;
    delta : LREAL;
  END_VAR
                  pointRelative := THIS^.processes.pointRelative.request(
    alphaUnits := alphaUnits,
    alpha := alpha,
    deltaUnits := deltaUnits,
    delta := delta);

                
END_METHOD

{attribute 'TcRpcEnable' := '1'}
METHOD stop : RequestResults
                  stop := THIS^.processes.stop.request();

                
END_METHOD

{attribute 'TcRpcEnable' := '1'}
METHOD quickStop : RequestResults
                  quickStop := THIS^.processes.quickStop.request();

                
END_METHOD

{attribute 'TcRpcEnable' := '1'}
METHOD powerOn : RequestResults
  VAR_INPUT
    azi : BOOL;
    ele : BOOL;
    roc : BOOL;
    ron : BOOL;
    fw : BOOL;
  END_VAR
                  powerOn := THIS^.processes.powerOn.request(
    azi := azi,
    ele := ele,
    roc := roc,
    ron := ron,
    fw := fw);

                
END_METHOD

{attribute 'TcRpcEnable' := '1'}
METHOD powerOff : RequestResults
                  powerOff := THIS^.processes.powerOff.request();

                
END_METHOD

{attribute 'TcRpcEnable' := '1'}
METHOD doHoming : RequestResults
                  doHoming := THIS^.processes.doHoming.request();

                
END_METHOD

{attribute 'TcRpcEnable' := '1'}
METHOD moveAbsolute : RequestResults
  VAR_INPUT
    units : AxesMoveUnits;
    azi : LREAL;
    ele : LREAL;
    rot : LREAL;
    roc : LREAL;
    ron : LREAL;
    doAzi : BOOL;
    doEle : BOOL;
    doRot : BOOL;
    doRoc : BOOL;
    doRon : BOOL;
    preferMostTravel : BOOL;
  END_VAR
                  moveAbsolute := THIS^.processes.moveAbsolute.request(
    units := units,
    azi := azi,
    ele := ele,
    rot := rot,
    roc := roc,
    ron := ron,
    doAzi := doAzi,
    doEle := doEle,
    doRot := doRot,
    doRoc := doRoc,
    doRon := doRon,
    preferMostTravel := preferMostTravel);

                
END_METHOD

{attribute 'TcRpcEnable' := '1'}
METHOD moveRelative : RequestResults
  VAR_INPUT
    units : AxesMoveUnits;
    azi : LREAL;
    ele : LREAL;
    rot : LREAL;
    roc : LREAL;
    ron : LREAL;
    doAzi : BOOL;
    doEle : BOOL;
    doRot : BOOL;
    doRoc : BOOL;
    doRon : BOOL;
    preferMostTravel : BOOL;
  END_VAR
                  moveRelative := THIS^.processes.moveRelative.request(
    units := units,
    azi := azi,
    ele := ele,
    rot := rot,
    roc := roc,
    ron := ron,
    doAzi := doAzi,
    doEle := doEle,
    doRot := doRot,
    doRoc := doRoc,
    doRon := doRon,
    preferMostTravel := preferMostTravel);

                
END_METHOD

{attribute 'TcRpcEnable' := '1'}
METHOD moveKnownPosition : RequestResults
  VAR_INPUT
    name : STRING;
  END_VAR
                  moveKnownPosition := THIS^.processes.moveKnownPosition.request( name := name );

                
END_METHOD

{attribute 'TcRpcEnable' := '1'}
METHOD enablePointingModel : RequestResults
  VAR_INPUT
    name : STRING;
  END_VAR
                  enablePointingModel := THIS^.processes.enablePointingModel.request( name := name );

                
END_METHOD

{attribute 'TcRpcEnable' := '1'}
METHOD disablePointingModel : RequestResults
                  disablePointingModel := THIS^.processes.disablePointingModel.request();

                
END_METHOD

{attribute 'TcRpcEnable' := '1'}
METHOD setAlphaDeltaVelocity : RequestResults
  VAR_INPUT
    units : AxesMoveVelocityUnits;
    alphaVelocity : LREAL;
    deltaVelocity : LREAL;
  END_VAR
                  setAlphaDeltaVelocity := THIS^.processes.setAlphaDeltaVelocity.request(
    units := units,
    alphaVelocity := alphaVelocity,
    deltaVelocity := deltaVelocity);

                
END_METHOD

{attribute 'TcRpcEnable' := '1'}
METHOD _log : BOOL
  VAR_INPUT
    name : STRING;  (* Name of this function block instance *)
  END_VAR
  VAR_IN_OUT
    buffer : LogBuffer;  (* Buffer to write all logging to *)
  END_VAR
  VAR
    subBuffer : LogBuffer;  (* Temporary buffer to write logging by parts (sub-statemachines) to *)
  END_VAR
                  THIS^.parts.azi._log(
    name := 'azi',
    buffer := subBuffer);
THIS^.parts.ele._log(
    name := 'ele',
    buffer := subBuffer);
THIS^.parts.roc._log(
    name := 'roc',
    buffer := subBuffer);
THIS^.parts.ron._log(
    name := 'ron',
    buffer := subBuffer);
THIS^.parts.io._log(
    name := 'io',
    buffer := subBuffer);
THIS^.parts.configManager._log(
    name := 'configManager',
    buffer := subBuffer);
THIS^.parts.tpoint._log(
    name := 'tpoint',
    buffer := subBuffer);
LOGGER(
    name := name,
    actualStatus := THIS^.actualStatus,
    previousStatus := THIS^.previousStatus,
    buffer := buffer,
    subBuffer := subBuffer,
    pHealthStatus := ADR(THIS^.statuses.healthStatus),
    pBusyStatus := ADR(THIS^.statuses.busyStatus));

                
END_METHOD
END_FUNCTION_BLOCK

FUNCTION_BLOCK SM_AxesTarget
  VAR_INPUT
    {attribute 'OPC.UA.DA' := '1'}
    {attribute 'OPC.UA.DA.Access' := '1'}
    isGiven : BOOL;  (* True if the target is given, false if not *)
    {attribute 'OPC.UA.DA' := '1'}
    {attribute 'OPC.UA.DA.Access' := '1'}
    isValid : BOOL;  (* True if the target is valid, false if not *)
    {attribute 'OPC.UA.DA' := '1'}
    {attribute 'OPC.UA.DA.Access' := '1'}
    isTooLow : BOOL;  (* True if the target is too low to calculate, false if not *)
    {attribute 'OPC.UA.DA' := '1'}
    {attribute 'OPC.UA.DA.Access' := '1'}
    alpha : AngularPosition;  (* The alpha coordinate (Right Ascention) *)
    {attribute 'OPC.UA.DA' := '1'}
    {attribute 'OPC.UA.DA.Access' := '1'}
    delta : AngularPosition;  (* The delta coordinate (Declination) *)
    {attribute 'OPC.UA.DA' := '1'}
    {attribute 'OPC.UA.DA.Access' := '1'}
    muAlpha : LREAL;  (* Right ascention proper motion, in arcseconds/year (not multiplied by cos(delta)!) *)
    {attribute 'OPC.UA.DA' := '1'}
    {attribute 'OPC.UA.DA.Access' := '1'}
    muDelta : LREAL;  (* Declination proper motion, in arcseconds/year *)
    {attribute 'OPC.UA.DA' := '1'}
    {attribute 'OPC.UA.DA.Access' := '1'}
    parallax : LREAL;  (* Object parallax, in arcseconds *)
    {attribute 'OPC.UA.DA' := '1'}
    {attribute 'OPC.UA.DA.Access' := '1'}
    radialVelocity : LREAL;  (* Object radial velocity, in km/s *)
    {attribute 'OPC.UA.DA' := '1'}
    {attribute 'OPC.UA.DA.Access' := '1'}
    epoch : LREAL;  (* Epoch, e.g. 2000.0 *)
    {attribute 'OPC.UA.DA' := '1'}
    {attribute 'OPC.UA.DA.Access' := '1'}
    alphaVelocity : AngularVelocity;  (* Additional target velocity (e.g. for solar system objects) in alpha direction *)
    {attribute 'OPC.UA.DA' := '1'}
    {attribute 'OPC.UA.DA.Access' := '1'}
    deltaVelocity : AngularVelocity;  (* Additional target velocity (e.g. for solar system objects) in delta direction *)
    {attribute 'OPC.UA.DA' := '1'}
    {attribute 'OPC.UA.DA.Access' := '1'}
    alphaTravelled : AngularPosition;  (* Alpha traveled so far due to the alphaVelocity *)
    {attribute 'OPC.UA.DA' := '1'}
    {attribute 'OPC.UA.DA.Access' := '1'}
    deltaTravelled : AngularPosition;  (* Delta traveled so far due to the deltaVelocity *)
    {attribute 'OPC.UA.DA' := '1'}
    {attribute 'OPC.UA.DA.Access' := '1'}
    alphaOffsetted : AngularPosition;  (* Alpha offsetted so far due to the alphaOffset *)
    {attribute 'OPC.UA.DA' := '1'}
    {attribute 'OPC.UA.DA.Access' := '1'}
    deltaOffsetted : AngularPosition;  (* Delta offsetted so far due to the deltaOffset *)
    {attribute 'OPC.UA.DA' := '1'}
    {attribute 'OPC.UA.DA.Access' := '1'}
    alphaStart : AngularPosition;  (* Original alpha without traveling (=alpha - alphaTraveled - alphaOffsetted) *)
    {attribute 'OPC.UA.DA' := '1'}
    {attribute 'OPC.UA.DA.Access' := '1'}
    deltaStart : AngularPosition;  (* Original delta without traveling (=delta - deltaTraveled - deltaOffsetted) *)
    {attribute 'OPC.UA.DA' := '1'}
    {attribute 'OPC.UA.DA.Access' := '1'}
    aziPos : AngularPosition;  (* The azimuth target position, as calculated by SLALIBl *)
    {attribute 'OPC.UA.DA' := '1'}
    {attribute 'OPC.UA.DA.Access' := '1'}
    aziVelo : AngularVelocity;  (* The azimuth target velocity, as calculated by SLALIB *)
    {attribute 'OPC.UA.DA' := '1'}
    {attribute 'OPC.UA.DA.Access' := '1'}
    aziAcc : AngularAcceleration;  (* The azimuth target acceleration, as calculated by SLALIB *)
    {attribute 'OPC.UA.DA' := '1'}
    {attribute 'OPC.UA.DA.Access' := '1'}
    elePos : AngularPosition;  (* The elevation target position, as calculated by SLALIB *)
    {attribute 'OPC.UA.DA' := '1'}
    {attribute 'OPC.UA.DA.Access' := '1'}
    eleVelo : AngularVelocity;  (* The elevation target velocity, as calculated by SLALIB *)
    {attribute 'OPC.UA.DA' := '1'}
    {attribute 'OPC.UA.DA.Access' := '1'}
    eleAcc : AngularAcceleration;  (* The elevation target acceleration, as calculated by SLALIB *)
    {attribute 'OPC.UA.DA' := '1'}
    {attribute 'OPC.UA.DA.Access' := '1'}
    paPos : AngularPosition;  (* The position angle target position, as calculated by SLALIB *)
    {attribute 'OPC.UA.DA' := '1'}
    {attribute 'OPC.UA.DA.Access' := '1'}
    paVelo : AngularVelocity;  (* The position angle target velocity, as calculated by SLALIB *)
    {attribute 'OPC.UA.DA' := '1'}
    {attribute 'OPC.UA.DA.Access' := '1'}
    paAcc : AngularAcceleration;  (* The position angle target acceleration, as calculated by SLALIB *)
    {attribute 'OPC.UA.DA' := '1'}
    {attribute 'OPC.UA.DA.Access' := '1'}
    aziPointingModelOffset : AngularPosition;  (* The azimuth pointing model offset calculated by the TPoint model *)
    {attribute 'OPC.UA.DA' := '1'}
    {attribute 'OPC.UA.DA.Access' := '1'}
    elePointingModelOffset : AngularPosition;  (* The elevation pointing model offset calculated by the TPoint model *)
    {attribute 'OPC.UA.DA' := '1'}
    {attribute 'OPC.UA.DA.Access' := '1'}
    correctedAzi : AngularPosition;  (* The azimuth target position, as calculated by SLALIB, corrected by the TPoint model *)
    {attribute 'OPC.UA.DA' := '1'}
    {attribute 'OPC.UA.DA.Access' := '1'}
    correctedEle : AngularPosition;  (* The elevation target position, as calculated by SLALIB, corrected by the TPoint model *)
  END_VAR
  VAR_OUTPUT
    {attribute 'OPC.UA.DA' := '1'}
    {attribute 'OPC.UA.DA.Access' := '1'}
    actualStatus : STRING;  (* Current status description *)
    previousStatus : STRING;  (* Previous status description *)
    statuses : AxesTargetStatuses;  (* Statuses of the state machine *)
  END_VAR

            statuses.healthStatus( isGood := isValid OR (NOT(isGiven)) );

          

{attribute 'TcRpcEnable' := '1'}
METHOD _log : BOOL
  VAR_INPUT
    name : STRING;  (* Name of this function block instance *)
  END_VAR
  VAR_IN_OUT
    buffer : LogBuffer;  (* Buffer to write all logging to *)
  END_VAR
  VAR
    subBuffer : LogBuffer;  (* Temporary buffer to write logging by parts (sub-statemachines) to *)
  END_VAR
                  LOGGER(
    name := name,
    actualStatus := THIS^.actualStatus,
    previousStatus := THIS^.previousStatus,
    buffer := buffer,
    subBuffer := subBuffer,
    pHealthStatus := ADR(THIS^.statuses.healthStatus));

                
END_METHOD
END_FUNCTION_BLOCK

FUNCTION_BLOCK SM_AxesFeedback
  VAR_INPUT
    {attribute 'OPC.UA.DA' := '1'}
    {attribute 'OPC.UA.DA.Access' := '1'}
    isValid : BOOL;  (* True if the feedback is valid, false if not *)
    {attribute 'OPC.UA.DA' := '1'}
    {attribute 'OPC.UA.DA.Access' := '1'}
    isTooLow : BOOL;  (* True if the feedback is too low to calculate, false if not *)
    {attribute 'OPC.UA.DA' := '1'}
    {attribute 'OPC.UA.DA.Access' := '1'}
    alpha : AngularPosition;  (* The alpha coordinate (Right Ascention) *)
    {attribute 'OPC.UA.DA' := '1'}
    {attribute 'OPC.UA.DA.Access' := '1'}
    delta : AngularPosition;  (* The delta coordinate (Declination) *)
    {attribute 'OPC.UA.DA' := '1'}
    {attribute 'OPC.UA.DA.Access' := '1'}
    aziPos : AngularPosition;  (* The measured AZI position, corrected by TPoint, and normalized to [0..2*PI] *)
    {attribute 'OPC.UA.DA' := '1'}
    {attribute 'OPC.UA.DA.Access' := '1'}
    elePos : AngularPosition;  (* The measured ELE position, corrected by TPoint, normalized to [-PI..PI] *)
    {attribute 'OPC.UA.DA' := '1'}
    {attribute 'OPC.UA.DA.Access' := '1'}
    rocPos : AngularPosition;  (* The measured ROC position, normalized to [-PI..PI] *)
    {attribute 'OPC.UA.DA' := '1'}
    {attribute 'OPC.UA.DA.Access' := '1'}
    ronPos : AngularPosition;  (* The measured RON position, normalized to [-PI..PI] *)
    {attribute 'OPC.UA.DA' := '1'}
    {attribute 'OPC.UA.DA.Access' := '1'}
    rotPos : AngularPosition;  (* The measured position of the currently active rotator (ROC or RON), normalized to [-PI..PI] *)
    {attribute 'OPC.UA.DA' := '1'}
    {attribute 'OPC.UA.DA.Access' := '1'}
    rotOffset : AngularPosition;  (* The active rotator offset, to North *)
    {attribute 'OPC.UA.DA' := '1'}
    {attribute 'OPC.UA.DA.Access' := '1'}
    rocOffset : AngularPosition;  (* The cassegrain rotator offset, to North *)
    {attribute 'OPC.UA.DA' := '1'}
    {attribute 'OPC.UA.DA.Access' := '1'}
    ronOffset : AngularPosition;  (* The nasmyth rotator offset, to North *)
  END_VAR
  VAR_OUTPUT
    {attribute 'OPC.UA.DA' := '1'}
    {attribute 'OPC.UA.DA.Access' := '1'}
    actualStatus : STRING;  (* Current status description *)
    previousStatus : STRING;  (* Previous status description *)
    statuses : AxesFeedbackStatuses;  (* Statuses of the state machine *)
  END_VAR

            statuses.healthStatus( isGood := isValid );

          

{attribute 'TcRpcEnable' := '1'}
METHOD _log : BOOL
  VAR_INPUT
    name : STRING;  (* Name of this function block instance *)
  END_VAR
  VAR_IN_OUT
    buffer : LogBuffer;  (* Buffer to write all logging to *)
  END_VAR
  VAR
    subBuffer : LogBuffer;  (* Temporary buffer to write logging by parts (sub-statemachines) to *)
  END_VAR
                  LOGGER(
    name := name,
    actualStatus := THIS^.actualStatus,
    previousStatus := THIS^.previousStatus,
    buffer := buffer,
    subBuffer := subBuffer,
    pHealthStatus := ADR(THIS^.statuses.healthStatus));

                
END_METHOD
END_FUNCTION_BLOCK

FUNCTION_BLOCK SM_AxesAzimuthAxis
  VAR_INPUT
    {attribute 'OPC.UA.DA' := '1'}
    {attribute 'OPC.UA.DA.Access' := '1'}
    id : AxesIds;  (* Id of this axis *)
    {attribute 'OPC.UA.DA' := '0'}
    isEnabled : BOOL;  (* Is control enabled? *)
    {attribute 'OPC.UA.DA' := '0'}
    REDUCTION_AZI_TO_TEL : LREAL := 1440.0;  (* The mechanical reduction between absolute encoder and telescope *)
    {attribute 'OPC.UA.DA' := '0'}
    REDUCTION_ABL_TO_TEL : LREAL := 180.0;  (* The mechanical reduction between absolute encoder and telescope *)
    {attribute 'OPC.UA.DA' := '0'}
    REDUCTION_ABS_ENC_TO_TEL : LREAL := 18.0;  (* The mechanical reduction between absolute encoder and telescope *)
  END_VAR
  VAR_OUTPUT
    {attribute 'OPC.UA.DA' := '1'}
    {attribute 'OPC.UA.DA.Access' := '1'}
    actualStatus : STRING;  (* Current status description *)
    previousStatus : STRING;  (* Previous status description *)
    {attribute 'OPC.UA.DA' := '1'}
    {attribute 'OPC.UA.DA.Access' := '1'}
    slipError : BOOL;  (* TRUE if the motor appears to be slipping w.r.t. the external encoder *)
    {attribute 'OPC.UA.DA' := '1'}
    {attribute 'OPC.UA.DA.Access' := '1'}
    positiveLimitSwitchError : BOOL;  (* TRUE if the positive limit switch has detected the axis *)
    {attribute 'OPC.UA.DA' := '1'}
    {attribute 'OPC.UA.DA.Access' := '1'}
    negativeLimitSwitchError : BOOL;  (* TRUE if the negative limit switch has detected the axis *)
    {attribute 'OPC.UA.DA' := '1'}
    {attribute 'OPC.UA.DA.Access' := '1'}
    setPosLimitReached : BOOL;  (* TRUE if the setpoint position has reached its limit *)
    {attribute 'OPC.UA.DA' := '1'}
    {attribute 'OPC.UA.DA.Access' := '1'}
    deviation1SecAverage : AngularPosition;  (* The deviation between target position and actual position, as a 1 second moving average *)
    {attribute 'OPC.UA.DA' := '1'}
    {attribute 'OPC.UA.DA.Access' := '1'}
    deviation1SecRMS : AngularPosition;  (* The deviation between target position and actual position, as a 1 second moving RMS error *)
    {attribute 'OPC.UA.DA' := '1'}
    {attribute 'OPC.UA.DA.Access' := '1'}
    targetPos : AngularPosition;  (* The target position *)
    {attribute 'OPC.UA.DA' := '1'}
    {attribute 'OPC.UA.DA.Access' := '1'}
    targetOffset : AngularPosition;  (* Cumulative offset of targetPos. Equals targetPos - targetStart *)
    {attribute 'OPC.UA.DA' := '1'}
    {attribute 'OPC.UA.DA.Access' := '1'}
    targetStart : AngularPosition;  (* Last absolute movement end position of the axis *)
    {attribute 'OPC.UA.DA' := '1'}
    {attribute 'OPC.UA.DA.Access' := '1'}
    setPos : AngularPosition;  (* The setpoint position (same as parts.physicalAxis!) *)
    {attribute 'OPC.UA.DA' := '1'}
    {attribute 'OPC.UA.DA.Access' := '1'}
    setVelo : AngularVelocity;  (* The setpoint velocity (same as parts.physicalAxis!) *)
    {attribute 'OPC.UA.DA' := '1'}
    {attribute 'OPC.UA.DA.Access' := '1'}
    setAcc : AngularAcceleration;  (* The setpoint acceleration (same as parts.physicalAxis!) *)
    {attribute 'OPC.UA.DA' := '1'}
    {attribute 'OPC.UA.DA.Access' := '1'}
    actPos : AngularPosition;  (* The actual position (same as parts.physicalAxis!) *)
    {attribute 'OPC.UA.DA' := '1'}
    {attribute 'OPC.UA.DA.Access' := '1'}
    actVelo : AngularVelocity;  (* The actual velocity (same as parts.physicalAxis!) *)
    {attribute 'OPC.UA.DA' := '1'}
    {attribute 'OPC.UA.DA.Access' := '1'}
    actAcc : AngularAcceleration;  (* The actual acceleration (same as parts.physicalAxis!) *)
    {attribute 'OPC.UA.DA' := '1'}
    {attribute 'OPC.UA.DA.Access' := '1'}
    actTorqueAzi : Torque;  (* The actual torque on the telescope axis by the AZI motor *)
    {attribute 'OPC.UA.DA' := '1'}
    {attribute 'OPC.UA.DA.Access' := '1'}
    actTorqueAbl : Torque;  (* The actual torque on the telescope axis by the ABL motor *)
    {attribute 'OPC.UA.DA' := '1'}
    {attribute 'OPC.UA.DA.Access' := '1'}
    lida1Position : AngularPosition;  (* Position of the telescope according to LIDA encoder no. 1 *)
    {attribute 'OPC.UA.DA' := '1'}
    {attribute 'OPC.UA.DA.Access' := '1'}
    lida2Position : AngularPosition;  (* Position of the telescope according to LIDA encoder no. 2 *)
    {attribute 'OPC.UA.DA' := '1'}
    {attribute 'OPC.UA.DA.Access' := '1'}
    lida3Position : AngularPosition;  (* Position of the telescope according to LIDA encoder no. 3 *)
    {attribute 'OPC.UA.DA' := '1'}
    {attribute 'OPC.UA.DA.Access' := '1'}
    lida4Position : AngularPosition;  (* Position of the telescope according to LIDA encoder no. 4 *)
    {attribute 'OPC.UA.DA' := '1'}
    {attribute 'OPC.UA.DA.Access' := '1'}
    lidaAveragePosition : AngularPosition;  (* Position of the telescope according to the average of the LIDA encoders *)
    {attribute 'OPC.UA.DA' := '1'}
    {attribute 'OPC.UA.DA.Access' := '1'}
    absoluteEncoderPosition : AngularPosition;  (* The position of the axis, based on the absolute encoder *)
    statuses : AxesAzimuthAxisStatuses;  (* Statuses of the state machine *)
    parts : AxesAzimuthAxisParts;  (* Parts of the state machine *)
    processes : AxesAzimuthAxisProcesses;  (* Processes of the state machine *)
  END_VAR
  VAR_IN_OUT
    {attribute 'OPC.UA.DA' := '0'}
    config : AxesAzimuthConfig;  (* Reference to the azimuth config *)
    {attribute 'OPC.UA.DA' := '0'}
    aziDriveChannel : AX52XXDriveChannel;  (* Reference to the AZI drive channel *)
    {attribute 'OPC.UA.DA' := '0'}
    ablDriveChannel : AX52XXDriveChannel;  (* Reference to the ABL drive channel *)
    {attribute 'OPC.UA.DA' := '0'}
    aziMainDriveChannel : AX52XXDriveChannel;  (* Reference to the main drive channel (channel A) of the drive *)
    {attribute 'OPC.UA.DA' := '0'}
    ablMainDriveChannel : AX52XXDriveChannel;  (* Reference to the main drive channel (channel A) of the drive *)
  END_VAR

            parts.virtualAxis( isEnabled := isEnabled );
parts.physicalAxis( isEnabled := isEnabled );
parts.ablAxis( isEnabled := isEnabled );
parts.lida1( isEnabled := isEnabled );
parts.lida2( isEnabled := isEnabled );
parts.lida3( isEnabled := isEnabled );
parts.lida4( isEnabled := isEnabled );
parts.absoluteEncoder();
statuses.busyStatus( isBusy := aziDriveChannel.statuses.busyStatus.busy OR (ablDriveChannel.statuses.busyStatus.busy OR (parts.virtualAxis.statuses.busyStatus.busy OR (parts.physicalAxis.statuses.busyStatus.busy OR (parts.ablAxis.statuses.busyStatus.busy OR (parts.lida1.statuses.busyStatus.busy OR (parts.lida2.statuses.busyStatus.busy OR (parts.lida3.statuses.busyStatus.busy OR (parts.lida4.statuses.busyStatus.busy OR (processes.moveAbsolute.statuses.busyStatus.busy OR (processes.moveRelative.statuses.busyStatus.busy OR (processes.moveVelocity.statuses.busyStatus.busy OR (processes.reset.statuses.busyStatus.busy OR (processes.moveOutOfLimitSwitch.statuses.busyStatus.busy OR (processes.powerOn.statuses.busyStatus.busy OR (processes.powerOff.statuses.busyStatus.busy OR (processes.doHoming.statuses.busyStatus.busy OR (processes.stop.statuses.busyStatus.busy OR (processes.quickStop.statuses.busyStatus.busy OR (processes.unlockBrake.statuses.busyStatus.busy OR processes.setPosition.statuses.busyStatus.busy))))))))))))))))))) );
statuses.healthStatus(
    isGood := (aziDriveChannel.statuses.healthStatus.isGood AND (ablDriveChannel.statuses.healthStatus.isGood AND (parts.virtualAxis.statuses.healthStatus.isGood AND (parts.physicalAxis.statuses.healthStatus.isGood AND (parts.ablAxis.statuses.healthStatus.isGood AND (parts.lida1.statuses.healthStatus.isGood AND (parts.lida2.statuses.healthStatus.isGood AND (parts.lida3.statuses.healthStatus.isGood AND (parts.lida4.statuses.healthStatus.isGood AND (parts.absoluteEncoder.statuses.healthStatus.isGood AND (processes.moveAbsolute.statuses.healthStatus.isGood AND (processes.moveRelative.statuses.healthStatus.isGood AND (processes.moveVelocity.statuses.healthStatus.isGood AND (processes.reset.statuses.healthStatus.isGood AND (processes.moveOutOfLimitSwitch.statuses.healthStatus.isGood AND (processes.powerOn.statuses.healthStatus.isGood AND (processes.powerOff.statuses.healthStatus.isGood AND (processes.doHoming.statuses.healthStatus.isGood AND (processes.stop.statuses.healthStatus.isGood AND (processes.quickStop.statuses.healthStatus.isGood AND (processes.unlockBrake.statuses.healthStatus.isGood AND processes.setPosition.statuses.healthStatus.isGood))))))))))))))))))))) AND ((NOT(slipError)) AND ((NOT(positiveLimitSwitchError)) AND (NOT(negativeLimitSwitchError)))),
    hasWarning := aziDriveChannel.statuses.healthStatus.hasWarning OR (ablDriveChannel.statuses.healthStatus.hasWarning OR (parts.virtualAxis.statuses.healthStatus.hasWarning OR (parts.physicalAxis.statuses.healthStatus.hasWarning OR (parts.ablAxis.statuses.healthStatus.hasWarning OR (parts.lida1.statuses.healthStatus.hasWarning OR (parts.lida2.statuses.healthStatus.hasWarning OR (parts.lida3.statuses.healthStatus.hasWarning OR (parts.lida4.statuses.healthStatus.hasWarning OR (parts.absoluteEncoder.statuses.healthStatus.hasWarning OR (processes.moveAbsolute.statuses.healthStatus.hasWarning OR (processes.moveRelative.statuses.healthStatus.hasWarning OR (processes.moveVelocity.statuses.healthStatus.hasWarning OR (processes.reset.statuses.healthStatus.hasWarning OR (processes.moveOutOfLimitSwitch.statuses.healthStatus.hasWarning OR (processes.powerOn.statuses.healthStatus.hasWarning OR (processes.powerOff.statuses.healthStatus.hasWarning OR (processes.doHoming.statuses.healthStatus.hasWarning OR (processes.stop.statuses.healthStatus.hasWarning OR (processes.quickStop.statuses.healthStatus.hasWarning OR (processes.unlockBrake.statuses.healthStatus.hasWarning OR processes.setPosition.statuses.healthStatus.hasWarning)))))))))))))))))))));
statuses.poweredStatus( isEnabled := parts.virtualAxis.statuses.poweredStatus.enabled AND (parts.physicalAxis.statuses.poweredStatus.enabled AND parts.ablAxis.statuses.poweredStatus.enabled) );
processes.moveAbsolute( isEnabled := isEnabled );
processes.moveRelative( isEnabled := isEnabled );
processes.moveVelocity( isEnabled := isEnabled );
processes.reset( isEnabled := isEnabled );
processes.moveOutOfLimitSwitch( isEnabled := isEnabled );
processes.powerOn( isEnabled := isEnabled );
processes.powerOff( isEnabled := isEnabled );
processes.doHoming( isEnabled := isEnabled );
processes.stop( isEnabled := isEnabled );
processes.quickStop( isEnabled := isEnabled );
processes.unlockBrake( isEnabled := isEnabled );
processes.setPosition( isEnabled := isEnabled );

          

{attribute 'TcRpcEnable' := '1'}
METHOD moveAbsolute : RequestResults
  VAR_INPUT
    units : AxesMoveUnits;
    value : LREAL;
    offset : LREAL;
  END_VAR
                  moveAbsolute := THIS^.processes.moveAbsolute.request(
    units := units,
    value := value,
    offset := offset);

                
END_METHOD

{attribute 'TcRpcEnable' := '1'}
METHOD moveRelative : RequestResults
  VAR_INPUT
    units : AxesMoveUnits;
    value : LREAL;
  END_VAR
                  moveRelative := THIS^.processes.moveRelative.request(
    units := units,
    value := value);

                
END_METHOD

{attribute 'TcRpcEnable' := '1'}
METHOD moveVelocity : RequestResults
  VAR_INPUT
    units : AxesMoveVelocityUnits;
    value : LREAL;
  END_VAR
                  moveVelocity := THIS^.processes.moveVelocity.request(
    units := units,
    value := value);

                
END_METHOD

{attribute 'TcRpcEnable' := '1'}
METHOD reset : RequestResults
                  reset := THIS^.processes.reset.request();

                
END_METHOD

{attribute 'TcRpcEnable' := '1'}
METHOD moveOutOfLimitSwitch : RequestResults
  VAR_INPUT
    switch : LimitSwitches;
  END_VAR
                  moveOutOfLimitSwitch := THIS^.processes.moveOutOfLimitSwitch.request( switch := switch );

                
END_METHOD

{attribute 'TcRpcEnable' := '1'}
METHOD powerOn : RequestResults
                  powerOn := THIS^.processes.powerOn.request();

                
END_METHOD

{attribute 'TcRpcEnable' := '1'}
METHOD powerOff : RequestResults
                  powerOff := THIS^.processes.powerOff.request();

                
END_METHOD

{attribute 'TcRpcEnable' := '1'}
METHOD doHoming : RequestResults
                  doHoming := THIS^.processes.doHoming.request();

                
END_METHOD

{attribute 'TcRpcEnable' := '1'}
METHOD stop : RequestResults
                  stop := THIS^.processes.stop.request();

                
END_METHOD

{attribute 'TcRpcEnable' := '1'}
METHOD quickStop : RequestResults
                  quickStop := THIS^.processes.quickStop.request();

                
END_METHOD

{attribute 'TcRpcEnable' := '1'}
METHOD unlockBrake : RequestResults
  VAR_INPUT
    seconds : LREAL;
  END_VAR
                  unlockBrake := THIS^.processes.unlockBrake.request( seconds := seconds );

                
END_METHOD

{attribute 'TcRpcEnable' := '1'}
METHOD setPosition : RequestResults
  VAR_INPUT
    value : LREAL;
  END_VAR
                  setPosition := THIS^.processes.setPosition.request( value := value );

                
END_METHOD

{attribute 'TcRpcEnable' := '1'}
METHOD _log : BOOL
  VAR_INPUT
    name : STRING;  (* Name of this function block instance *)
  END_VAR
  VAR_IN_OUT
    buffer : LogBuffer;  (* Buffer to write all logging to *)
  END_VAR
  VAR
    subBuffer : LogBuffer;  (* Temporary buffer to write logging by parts (sub-statemachines) to *)
  END_VAR
                  THIS^.parts.virtualAxis._log(
    name := 'virtualAxis',
    buffer := subBuffer);
THIS^.parts.physicalAxis._log(
    name := 'physicalAxis',
    buffer := subBuffer);
THIS^.parts.ablAxis._log(
    name := 'ablAxis',
    buffer := subBuffer);
THIS^.parts.lida1._log(
    name := 'lida1',
    buffer := subBuffer);
THIS^.parts.lida2._log(
    name := 'lida2',
    buffer := subBuffer);
THIS^.parts.lida3._log(
    name := 'lida3',
    buffer := subBuffer);
THIS^.parts.lida4._log(
    name := 'lida4',
    buffer := subBuffer);
THIS^.parts.absoluteEncoder._log(
    name := 'absoluteEncoder',
    buffer := subBuffer);
LOGGER(
    name := name,
    actualStatus := THIS^.actualStatus,
    previousStatus := THIS^.previousStatus,
    buffer := buffer,
    subBuffer := subBuffer,
    pHealthStatus := ADR(THIS^.statuses.healthStatus),
    pBusyStatus := ADR(THIS^.statuses.busyStatus));

                
END_METHOD
END_FUNCTION_BLOCK

FUNCTION_BLOCK SM_AxesElevationAxis
  VAR_INPUT
    {attribute 'OPC.UA.DA' := '1'}
    {attribute 'OPC.UA.DA.Access' := '1'}
    id : AxesIds;  (* Id of this axis *)
    {attribute 'OPC.UA.DA' := '0'}
    isEnabled : BOOL;  (* Is control enabled? *)
    {attribute 'OPC.UA.DA' := '0'}
    REDUCTION_MOT_TO_TEL : LREAL := 1440.0;  (* The mechanical reduction between absolute encoder and telescope *)
    {attribute 'OPC.UA.DA' := '0'}
    REDUCTION_ABS_ENC_TO_TEL : LREAL := 18.0;  (* The mechanical reduction between absolute encoder and telescope *)
  END_VAR
  VAR_OUTPUT
    {attribute 'OPC.UA.DA' := '1'}
    {attribute 'OPC.UA.DA.Access' := '1'}
    actualStatus : STRING;  (* Current status description *)
    previousStatus : STRING;  (* Previous status description *)
    {attribute 'OPC.UA.DA' := '1'}
    {attribute 'OPC.UA.DA.Access' := '1'}
    slipError : BOOL;  (* TRUE if the motor appears to be slipping w.r.t. the external encoder *)
    {attribute 'OPC.UA.DA' := '1'}
    {attribute 'OPC.UA.DA.Access' := '1'}
    positiveLimitSwitchError : BOOL;  (* TRUE if the positive limit switch has detected the axis *)
    {attribute 'OPC.UA.DA' := '1'}
    {attribute 'OPC.UA.DA.Access' := '1'}
    negativeLimitSwitchError : BOOL;  (* TRUE if the negative limit switch has detected the axis *)
    {attribute 'OPC.UA.DA' := '1'}
    {attribute 'OPC.UA.DA.Access' := '1'}
    setPosLimitReached : BOOL;  (* TRUE if the setpoint position has reached its limit *)
    {attribute 'OPC.UA.DA' := '1'}
    {attribute 'OPC.UA.DA.Access' := '1'}
    deviation1SecAverage : AngularPosition;  (* The deviation between target position and actual position, as a 1 second moving average *)
    {attribute 'OPC.UA.DA' := '1'}
    {attribute 'OPC.UA.DA.Access' := '1'}
    deviation1SecRMS : AngularPosition;  (* The deviation between target position and actual position, as a 1 second moving RMS error *)
    {attribute 'OPC.UA.DA' := '1'}
    {attribute 'OPC.UA.DA.Access' := '1'}
    targetPos : AngularPosition;  (* The target position *)
    {attribute 'OPC.UA.DA' := '1'}
    {attribute 'OPC.UA.DA.Access' := '1'}
    targetOffset : AngularPosition;  (* Cumulative offset of targetPos. Equals targetPos - targetStart *)
    {attribute 'OPC.UA.DA' := '1'}
    {attribute 'OPC.UA.DA.Access' := '1'}
    targetStart : AngularPosition;  (* Last absolute movement end position of the axis *)
    {attribute 'OPC.UA.DA' := '1'}
    {attribute 'OPC.UA.DA.Access' := '1'}
    setPos : AngularPosition;  (* The setpoint position (same as parts.physicalAxis!) *)
    {attribute 'OPC.UA.DA' := '1'}
    {attribute 'OPC.UA.DA.Access' := '1'}
    setVelo : AngularVelocity;  (* The setpoint velocity (same as parts.physicalAxis!) *)
    {attribute 'OPC.UA.DA' := '1'}
    {attribute 'OPC.UA.DA.Access' := '1'}
    setAcc : AngularAcceleration;  (* The setpoint acceleration (same as parts.physicalAxis!) *)
    {attribute 'OPC.UA.DA' := '1'}
    {attribute 'OPC.UA.DA.Access' := '1'}
    actPos : AngularPosition;  (* The actual position (same as parts.physicalAxis!) *)
    {attribute 'OPC.UA.DA' := '1'}
    {attribute 'OPC.UA.DA.Access' := '1'}
    actVelo : AngularVelocity;  (* The actual velocity (same as parts.physicalAxis!) *)
    {attribute 'OPC.UA.DA' := '1'}
    {attribute 'OPC.UA.DA.Access' := '1'}
    actAcc : AngularAcceleration;  (* The actual acceleration (same as parts.physicalAxis!) *)
    {attribute 'OPC.UA.DA' := '1'}
    {attribute 'OPC.UA.DA.Access' := '1'}
    actTorque : Torque;  (* The actual torque on the telescope axis by the ELE motor *)
    {attribute 'OPC.UA.DA' := '1'}
    {attribute 'OPC.UA.DA.Access' := '1'}
    lida1Position : AngularPosition;  (* Position of the telescope according to LIDA encoder no. 1 *)
    {attribute 'OPC.UA.DA' := '1'}
    {attribute 'OPC.UA.DA.Access' := '1'}
    lida2Position : AngularPosition;  (* Position of the telescope according to LIDA encoder no. 2 *)
    {attribute 'OPC.UA.DA' := '1'}
    {attribute 'OPC.UA.DA.Access' := '1'}
    lidaAveragePosition : AngularPosition;  (* Position of the telescope according to the average of the LIDA encoders *)
    {attribute 'OPC.UA.DA' := '1'}
    {attribute 'OPC.UA.DA.Access' := '1'}
    absoluteEncoderPosition : AngularPosition;  (* Position of the telescope according to the absolute encoder *)
    statuses : AxesElevationAxisStatuses;  (* Statuses of the state machine *)
    parts : AxesElevationAxisParts;  (* Parts of the state machine *)
    processes : AxesElevationAxisProcesses;  (* Processes of the state machine *)
  END_VAR
  VAR_IN_OUT
    {attribute 'OPC.UA.DA' := '0'}
    config : AxesElevationConfig;  (* Reference to the elevation config *)
    {attribute 'OPC.UA.DA' := '0'}
    driveChannel : AX52XXDriveChannel;  (* Reference to the ELE drive channel *)
    {attribute 'OPC.UA.DA' := '0'}
    mainDriveChannel : AX52XXDriveChannel;  (* Reference to the main drive channel (channel A) of the drive *)
  END_VAR

            parts.virtualAxis( isEnabled := isEnabled );
parts.physicalAxis( isEnabled := isEnabled );
parts.lida1( isEnabled := isEnabled );
parts.lida2( isEnabled := isEnabled );
parts.absoluteEncoder();
statuses.busyStatus( isBusy := driveChannel.statuses.busyStatus.busy OR (parts.virtualAxis.statuses.busyStatus.busy OR (parts.physicalAxis.statuses.busyStatus.busy OR (parts.lida1.statuses.busyStatus.busy OR (parts.lida2.statuses.busyStatus.busy OR (processes.moveAbsolute.statuses.busyStatus.busy OR (processes.moveRelative.statuses.busyStatus.busy OR (processes.moveVelocity.statuses.busyStatus.busy OR (processes.reset.statuses.busyStatus.busy OR (processes.moveOutOfLimitSwitch.statuses.busyStatus.busy OR (processes.powerOn.statuses.busyStatus.busy OR (processes.powerOff.statuses.busyStatus.busy OR (processes.doHoming.statuses.busyStatus.busy OR (processes.stop.statuses.busyStatus.busy OR (processes.quickStop.statuses.busyStatus.busy OR (processes.unlockBrake.statuses.busyStatus.busy OR processes.setPosition.statuses.busyStatus.busy))))))))))))))) );
statuses.healthStatus(
    isGood := (driveChannel.statuses.healthStatus.isGood AND (parts.virtualAxis.statuses.healthStatus.isGood AND (parts.physicalAxis.statuses.healthStatus.isGood AND (parts.lida1.statuses.healthStatus.isGood AND (parts.lida2.statuses.healthStatus.isGood AND (parts.absoluteEncoder.statuses.healthStatus.isGood AND (processes.moveAbsolute.statuses.healthStatus.isGood AND (processes.moveRelative.statuses.healthStatus.isGood AND (processes.moveVelocity.statuses.healthStatus.isGood AND (processes.reset.statuses.healthStatus.isGood AND (processes.moveOutOfLimitSwitch.statuses.healthStatus.isGood AND (processes.powerOn.statuses.healthStatus.isGood AND (processes.powerOff.statuses.healthStatus.isGood AND (processes.doHoming.statuses.healthStatus.isGood AND (processes.stop.statuses.healthStatus.isGood AND (processes.quickStop.statuses.healthStatus.isGood AND (processes.unlockBrake.statuses.healthStatus.isGood AND processes.setPosition.statuses.healthStatus.isGood))))))))))))))))) AND ((NOT(slipError)) AND ((NOT(positiveLimitSwitchError)) AND (NOT(negativeLimitSwitchError)))),
    hasWarning := driveChannel.statuses.healthStatus.hasWarning OR (parts.virtualAxis.statuses.healthStatus.hasWarning OR (parts.physicalAxis.statuses.healthStatus.hasWarning OR (parts.lida1.statuses.healthStatus.hasWarning OR (parts.lida2.statuses.healthStatus.hasWarning OR (parts.absoluteEncoder.statuses.healthStatus.hasWarning OR (processes.moveAbsolute.statuses.healthStatus.hasWarning OR (processes.moveRelative.statuses.healthStatus.hasWarning OR (processes.moveVelocity.statuses.healthStatus.hasWarning OR (processes.reset.statuses.healthStatus.hasWarning OR (processes.moveOutOfLimitSwitch.statuses.healthStatus.hasWarning OR (processes.powerOn.statuses.healthStatus.hasWarning OR (processes.powerOff.statuses.healthStatus.hasWarning OR (processes.doHoming.statuses.healthStatus.hasWarning OR (processes.stop.statuses.healthStatus.hasWarning OR (processes.quickStop.statuses.healthStatus.hasWarning OR (processes.unlockBrake.statuses.healthStatus.hasWarning OR processes.setPosition.statuses.healthStatus.hasWarning)))))))))))))))));
statuses.poweredStatus( isEnabled := parts.virtualAxis.statuses.poweredStatus.enabled AND parts.physicalAxis.statuses.poweredStatus.enabled );
processes.moveAbsolute( isEnabled := isEnabled );
processes.moveRelative( isEnabled := isEnabled );
processes.moveVelocity( isEnabled := isEnabled );
processes.reset( isEnabled := isEnabled );
processes.moveOutOfLimitSwitch( isEnabled := isEnabled );
processes.powerOn( isEnabled := isEnabled );
processes.powerOff( isEnabled := isEnabled );
processes.doHoming( isEnabled := isEnabled );
processes.stop( isEnabled := isEnabled );
processes.quickStop( isEnabled := isEnabled );
processes.setPosition( isEnabled := isEnabled );
processes.unlockBrake();

          

{attribute 'TcRpcEnable' := '1'}
METHOD moveAbsolute : RequestResults
  VAR_INPUT
    units : AxesMoveUnits;
    value : LREAL;
    offset : LREAL;
  END_VAR
                  moveAbsolute := THIS^.processes.moveAbsolute.request(
    units := units,
    value := value,
    offset := offset);

                
END_METHOD

{attribute 'TcRpcEnable' := '1'}
METHOD moveRelative : RequestResults
  VAR_INPUT
    units : AxesMoveUnits;
    value : LREAL;
  END_VAR
                  moveRelative := THIS^.processes.moveRelative.request(
    units := units,
    value := value);

                
END_METHOD

{attribute 'TcRpcEnable' := '1'}
METHOD moveVelocity : RequestResults
  VAR_INPUT
    units : AxesMoveVelocityUnits;
    value : LREAL;
  END_VAR
                  moveVelocity := THIS^.processes.moveVelocity.request(
    units := units,
    value := value);

                
END_METHOD

{attribute 'TcRpcEnable' := '1'}
METHOD reset : RequestResults
                  reset := THIS^.processes.reset.request();

                
END_METHOD

{attribute 'TcRpcEnable' := '1'}
METHOD moveOutOfLimitSwitch : RequestResults
  VAR_INPUT
    switch : LimitSwitches;
  END_VAR
                  moveOutOfLimitSwitch := THIS^.processes.moveOutOfLimitSwitch.request( switch := switch );

                
END_METHOD

{attribute 'TcRpcEnable' := '1'}
METHOD powerOn : RequestResults
                  powerOn := THIS^.processes.powerOn.request();

                
END_METHOD

{attribute 'TcRpcEnable' := '1'}
METHOD powerOff : RequestResults
                  powerOff := THIS^.processes.powerOff.request();

                
END_METHOD

{attribute 'TcRpcEnable' := '1'}
METHOD doHoming : RequestResults
                  doHoming := THIS^.processes.doHoming.request();

                
END_METHOD

{attribute 'TcRpcEnable' := '1'}
METHOD stop : RequestResults
                  stop := THIS^.processes.stop.request();

                
END_METHOD

{attribute 'TcRpcEnable' := '1'}
METHOD quickStop : RequestResults
                  quickStop := THIS^.processes.quickStop.request();

                
END_METHOD

{attribute 'TcRpcEnable' := '1'}
METHOD setPosition : RequestResults
  VAR_INPUT
    value : LREAL;
  END_VAR
                  setPosition := THIS^.processes.setPosition.request( value := value );

                
END_METHOD

{attribute 'TcRpcEnable' := '1'}
METHOD unlockBrake : RequestResults
  VAR_INPUT
    seconds : LREAL;
  END_VAR
                  unlockBrake := THIS^.processes.unlockBrake.request( seconds := seconds );

                
END_METHOD

{attribute 'TcRpcEnable' := '1'}
METHOD _log : BOOL
  VAR_INPUT
    name : STRING;  (* Name of this function block instance *)
  END_VAR
  VAR_IN_OUT
    buffer : LogBuffer;  (* Buffer to write all logging to *)
  END_VAR
  VAR
    subBuffer : LogBuffer;  (* Temporary buffer to write logging by parts (sub-statemachines) to *)
  END_VAR
                  THIS^.parts.virtualAxis._log(
    name := 'virtualAxis',
    buffer := subBuffer);
THIS^.parts.physicalAxis._log(
    name := 'physicalAxis',
    buffer := subBuffer);
THIS^.parts.lida1._log(
    name := 'lida1',
    buffer := subBuffer);
THIS^.parts.lida2._log(
    name := 'lida2',
    buffer := subBuffer);
THIS^.parts.absoluteEncoder._log(
    name := 'absoluteEncoder',
    buffer := subBuffer);
LOGGER(
    name := name,
    actualStatus := THIS^.actualStatus,
    previousStatus := THIS^.previousStatus,
    buffer := buffer,
    subBuffer := subBuffer,
    pHealthStatus := ADR(THIS^.statuses.healthStatus),
    pBusyStatus := ADR(THIS^.statuses.busyStatus));

                
END_METHOD
END_FUNCTION_BLOCK

FUNCTION_BLOCK SM_AxesRotationAxis
  VAR_INPUT
    {attribute 'OPC.UA.DA' := '1'}
    {attribute 'OPC.UA.DA.Access' := '1'}
    id : AxesIds;  (* Id of this axis *)
    {attribute 'OPC.UA.DA' := '0'}
    isEnabled : BOOL;  (* Is control enabled? *)
  END_VAR
  VAR_OUTPUT
    {attribute 'OPC.UA.DA' := '1'}
    {attribute 'OPC.UA.DA.Access' := '1'}
    actualStatus : STRING;  (* Current status description *)
    previousStatus : STRING;  (* Previous status description *)
    {attribute 'OPC.UA.DA' := '1'}
    {attribute 'OPC.UA.DA.Access' := '1'}
    positiveLimitSwitchError : BOOL;  (* TRUE if the positive limit switch has detected the axis *)
    {attribute 'OPC.UA.DA' := '1'}
    {attribute 'OPC.UA.DA.Access' := '1'}
    negativeLimitSwitchError : BOOL;  (* TRUE if the negative limit switch has detected the axis *)
    {attribute 'OPC.UA.DA' := '1'}
    {attribute 'OPC.UA.DA.Access' := '1'}
    setPosLimitReached : BOOL;  (* TRUE if the setpoint position has reached its limit *)
    {attribute 'OPC.UA.DA' := '1'}
    {attribute 'OPC.UA.DA.Access' := '1'}
    deviation1SecAverage : AngularPosition;  (* The deviation between target position and actual position, as a 1 second moving average *)
    {attribute 'OPC.UA.DA' := '1'}
    {attribute 'OPC.UA.DA.Access' := '1'}
    deviation1SecRMS : AngularPosition;  (* The deviation between target position and actual position, as a 1 second moving RMS error *)
    {attribute 'OPC.UA.DA' := '1'}
    {attribute 'OPC.UA.DA.Access' := '1'}
    targetPos : AngularPosition;  (* The target position *)
    {attribute 'OPC.UA.DA' := '1'}
    {attribute 'OPC.UA.DA.Access' := '1'}
    targetOffset : AngularPosition;  (* Cumulative offset of targetPos. Equals targetPos - targetStart *)
    {attribute 'OPC.UA.DA' := '1'}
    {attribute 'OPC.UA.DA.Access' := '1'}
    targetStart : AngularPosition;  (* Last absolute movement end position of the axis *)
    {attribute 'OPC.UA.DA' := '1'}
    {attribute 'OPC.UA.DA.Access' := '1'}
    setPos : AngularPosition;  (* The setpoint position (same as parts.physicalAxis!) *)
    {attribute 'OPC.UA.DA' := '1'}
    {attribute 'OPC.UA.DA.Access' := '1'}
    setVelo : AngularVelocity;  (* The setpoint velocity (same as parts.physicalAxis!) *)
    {attribute 'OPC.UA.DA' := '1'}
    {attribute 'OPC.UA.DA.Access' := '1'}
    setAcc : AngularAcceleration;  (* The setpoint acceleration (same as parts.physicalAxis!) *)
    {attribute 'OPC.UA.DA' := '1'}
    {attribute 'OPC.UA.DA.Access' := '1'}
    actPos : AngularPosition;  (* The actual position (same as parts.eleAxis!) *)
    {attribute 'OPC.UA.DA' := '1'}
    {attribute 'OPC.UA.DA.Access' := '1'}
    actVelo : AngularVelocity;  (* The actual velocity (same as parts.eleAxis!) *)
    {attribute 'OPC.UA.DA' := '1'}
    {attribute 'OPC.UA.DA.Access' := '1'}
    actAcc : AngularAcceleration;  (* The actual acceleration (same as parts.eleAxis!) *)
    {attribute 'OPC.UA.DA' := '1'}
    {attribute 'OPC.UA.DA.Access' := '1'}
    actTorque : Torque;  (* The actual torque on the telescope axis by the ELE motor *)
    statuses : AxesRotationAxisStatuses;  (* Statuses of the state machine *)
    parts : AxesRotationAxisParts;  (* Parts of the state machine *)
    processes : AxesRotationAxisProcesses;  (* Processes of the state machine *)
  END_VAR
  VAR_IN_OUT
    {attribute 'OPC.UA.DA' := '0'}
    config : AxesRotationConfig;  (* Reference to the rotation config *)
    {attribute 'OPC.UA.DA' := '0'}
    driveChannel : AX52XXDriveChannel;  (* Reference to the axis drive channel *)
    {attribute 'OPC.UA.DA' := '0'}
    mainDriveChannel : AX52XXDriveChannel;  (* Reference to the main drive channel (channel A) of the drive *)
  END_VAR

            parts.virtualAxis( isEnabled := isEnabled );
parts.physicalAxis( isEnabled := isEnabled );
statuses.busyStatus( isBusy := driveChannel.statuses.busyStatus.busy OR (parts.virtualAxis.statuses.busyStatus.busy OR (parts.physicalAxis.statuses.busyStatus.busy OR (processes.moveAbsolute.statuses.busyStatus.busy OR (processes.moveRelative.statuses.busyStatus.busy OR (processes.moveVelocity.statuses.busyStatus.busy OR (processes.reset.statuses.busyStatus.busy OR (processes.moveOutOfLimitSwitch.statuses.busyStatus.busy OR (processes.powerOn.statuses.busyStatus.busy OR (processes.powerOff.statuses.busyStatus.busy OR (processes.stop.statuses.busyStatus.busy OR (processes.quickStop.statuses.busyStatus.busy OR processes.setPosition.statuses.busyStatus.busy))))))))))) );
statuses.healthStatus(
    isGood := (driveChannel.statuses.healthStatus.isGood AND (parts.virtualAxis.statuses.healthStatus.isGood AND (parts.physicalAxis.statuses.healthStatus.isGood AND (processes.moveAbsolute.statuses.healthStatus.isGood AND (processes.moveRelative.statuses.healthStatus.isGood AND (processes.moveVelocity.statuses.healthStatus.isGood AND (processes.reset.statuses.healthStatus.isGood AND (processes.moveOutOfLimitSwitch.statuses.healthStatus.isGood AND (processes.powerOn.statuses.healthStatus.isGood AND (processes.powerOff.statuses.healthStatus.isGood AND (processes.stop.statuses.healthStatus.isGood AND (processes.quickStop.statuses.healthStatus.isGood AND processes.setPosition.statuses.healthStatus.isGood)))))))))))) AND ((NOT(positiveLimitSwitchError)) AND (NOT(negativeLimitSwitchError))),
    hasWarning := driveChannel.statuses.healthStatus.hasWarning OR (parts.virtualAxis.statuses.healthStatus.hasWarning OR (parts.physicalAxis.statuses.healthStatus.hasWarning OR (processes.moveAbsolute.statuses.healthStatus.hasWarning OR (processes.moveRelative.statuses.healthStatus.hasWarning OR (processes.moveVelocity.statuses.healthStatus.hasWarning OR (processes.reset.statuses.healthStatus.hasWarning OR (processes.moveOutOfLimitSwitch.statuses.healthStatus.hasWarning OR (processes.powerOn.statuses.healthStatus.hasWarning OR (processes.powerOff.statuses.healthStatus.hasWarning OR (processes.stop.statuses.healthStatus.hasWarning OR (processes.quickStop.statuses.healthStatus.hasWarning OR processes.setPosition.statuses.healthStatus.hasWarning))))))))))));
statuses.poweredStatus( isEnabled := parts.virtualAxis.statuses.poweredStatus.enabled AND parts.physicalAxis.statuses.poweredStatus.enabled );
processes.moveAbsolute( isEnabled := isEnabled );
processes.moveRelative( isEnabled := isEnabled );
processes.moveVelocity( isEnabled := isEnabled );
processes.reset( isEnabled := isEnabled );
processes.moveOutOfLimitSwitch( isEnabled := isEnabled );
processes.powerOn( isEnabled := isEnabled );
processes.powerOff( isEnabled := isEnabled );
processes.stop( isEnabled := isEnabled );
processes.quickStop( isEnabled := isEnabled );
processes.setPosition( isEnabled := isEnabled );

          

{attribute 'TcRpcEnable' := '1'}
METHOD moveAbsolute : RequestResults
  VAR_INPUT
    units : AxesMoveUnits;
    value : LREAL;
    offset : LREAL;
  END_VAR
                  moveAbsolute := THIS^.processes.moveAbsolute.request(
    units := units,
    value := value,
    offset := offset);

                
END_METHOD

{attribute 'TcRpcEnable' := '1'}
METHOD moveRelative : RequestResults
  VAR_INPUT
    units : AxesMoveUnits;
    value : LREAL;
  END_VAR
                  moveRelative := THIS^.processes.moveRelative.request(
    units := units,
    value := value);

                
END_METHOD

{attribute 'TcRpcEnable' := '1'}
METHOD moveVelocity : RequestResults
  VAR_INPUT
    units : AxesMoveVelocityUnits;
    value : LREAL;
  END_VAR
                  moveVelocity := THIS^.processes.moveVelocity.request(
    units := units,
    value := value);

                
END_METHOD

{attribute 'TcRpcEnable' := '1'}
METHOD reset : RequestResults
                  reset := THIS^.processes.reset.request();

                
END_METHOD

{attribute 'TcRpcEnable' := '1'}
METHOD moveOutOfLimitSwitch : RequestResults
  VAR_INPUT
    switch : LimitSwitches;
  END_VAR
                  moveOutOfLimitSwitch := THIS^.processes.moveOutOfLimitSwitch.request( switch := switch );

                
END_METHOD

{attribute 'TcRpcEnable' := '1'}
METHOD powerOn : RequestResults
                  powerOn := THIS^.processes.powerOn.request();

                
END_METHOD

{attribute 'TcRpcEnable' := '1'}
METHOD powerOff : RequestResults
                  powerOff := THIS^.processes.powerOff.request();

                
END_METHOD

{attribute 'TcRpcEnable' := '1'}
METHOD stop : RequestResults
                  stop := THIS^.processes.stop.request();

                
END_METHOD

{attribute 'TcRpcEnable' := '1'}
METHOD quickStop : RequestResults
                  quickStop := THIS^.processes.quickStop.request();

                
END_METHOD

{attribute 'TcRpcEnable' := '1'}
METHOD setPosition : RequestResults
  VAR_INPUT
    value : LREAL;
  END_VAR
                  setPosition := THIS^.processes.setPosition.request( value := value );

                
END_METHOD

{attribute 'TcRpcEnable' := '1'}
METHOD _log : BOOL
  VAR_INPUT
    name : STRING;  (* Name of this function block instance *)
  END_VAR
  VAR_IN_OUT
    buffer : LogBuffer;  (* Buffer to write all logging to *)
  END_VAR
  VAR
    subBuffer : LogBuffer;  (* Temporary buffer to write logging by parts (sub-statemachines) to *)
  END_VAR
                  THIS^.parts.virtualAxis._log(
    name := 'virtualAxis',
    buffer := subBuffer);
THIS^.parts.physicalAxis._log(
    name := 'physicalAxis',
    buffer := subBuffer);
LOGGER(
    name := name,
    actualStatus := THIS^.actualStatus,
    previousStatus := THIS^.previousStatus,
    buffer := buffer,
    subBuffer := subBuffer,
    pHealthStatus := ADR(THIS^.statuses.healthStatus),
    pBusyStatus := ADR(THIS^.statuses.busyStatus));

                
END_METHOD
END_FUNCTION_BLOCK

FUNCTION_BLOCK SM_AxesPointingModelSetup
  VAR_INPUT
    {attribute 'OPC.UA.DA' := '1'}
    {attribute 'OPC.UA.DA.Access' := '1'}
    editableConfig : AxesPointingModelConfig;  (* Editable configuration of the particular TPOINT model *)
    {attribute 'OPC.UA.DA' := '0'}
    isEnabled : BOOL;  (* Is control enabled? *)
  END_VAR
  VAR_OUTPUT
    {attribute 'OPC.UA.DA' := '1'}
    {attribute 'OPC.UA.DA.Access' := '1'}
    actualStatus : STRING;  (* Current status description *)
    previousStatus : STRING;  (* Previous status description *)
    {attribute 'OPC.UA.DA' := '1'}
    {attribute 'OPC.UA.DA.Access' := '1'}
    config : AxesPointingModelConfig;  (* Active configuration of the particular TPOINT model *)
    parts : AxesPointingModelSetupParts;  (* Parts of the state machine *)
  END_VAR

            parts.configManager( isEnabled := isEnabled );

          

{attribute 'TcRpcEnable' := '1'}
METHOD _log : BOOL
  VAR_INPUT
    name : STRING;  (* Name of this function block instance *)
  END_VAR
  VAR_IN_OUT
    buffer : LogBuffer;  (* Buffer to write all logging to *)
  END_VAR
  VAR
    subBuffer : LogBuffer;  (* Temporary buffer to write logging by parts (sub-statemachines) to *)
  END_VAR
                  THIS^.parts.configManager._log(
    name := 'configManager',
    buffer := subBuffer);
LOGGER(
    name := name,
    actualStatus := THIS^.actualStatus,
    previousStatus := THIS^.previousStatus,
    buffer := buffer,
    subBuffer := subBuffer);

                
END_METHOD
END_FUNCTION_BLOCK

FUNCTION_BLOCK SM_AxesPointingModelsSetup
  VAR_INPUT
    {attribute 'OPC.UA.DA' := '0'}
    isEnabled : BOOL;  (* Is control enabled? *)
  END_VAR
  VAR_OUTPUT
    {attribute 'OPC.UA.DA' := '1'}
    {attribute 'OPC.UA.DA.Access' := '1'}
    actualStatus : STRING;  (* Current status description *)
    previousStatus : STRING;  (* Previous status description *)
    statuses : AxesPointingModelsSetupStatuses;  (* Statuses of the state machine *)
    parts : AxesPointingModelsSetupParts;  (* Parts of the state machine *)
  END_VAR

            parts.model0( isEnabled := isEnabled );
parts.model1( isEnabled := isEnabled );
parts.model2( isEnabled := isEnabled );
parts.model3( isEnabled := isEnabled );
parts.model4( isEnabled := isEnabled );
parts.model5( isEnabled := isEnabled );
parts.model6( isEnabled := isEnabled );
parts.model7( isEnabled := isEnabled );
parts.model8( isEnabled := isEnabled );
parts.model9( isEnabled := isEnabled );
statuses.busyStatus( isBusy := parts.model0.parts.configManager.statuses.busyStatus.busy OR (parts.model1.parts.configManager.statuses.busyStatus.busy OR (parts.model2.parts.configManager.statuses.busyStatus.busy OR (parts.model3.parts.configManager.statuses.busyStatus.busy OR (parts.model4.parts.configManager.statuses.busyStatus.busy OR (parts.model5.parts.configManager.statuses.busyStatus.busy OR (parts.model6.parts.configManager.statuses.busyStatus.busy OR (parts.model7.parts.configManager.statuses.busyStatus.busy OR (parts.model8.parts.configManager.statuses.busyStatus.busy OR parts.model9.parts.configManager.statuses.busyStatus.busy)))))))) );
statuses.healthStatus(
    isGood := parts.model0.parts.configManager.statuses.healthStatus.isGood AND (parts.model1.parts.configManager.statuses.healthStatus.isGood AND (parts.model2.parts.configManager.statuses.healthStatus.isGood AND (parts.model3.parts.configManager.statuses.healthStatus.isGood AND (parts.model4.parts.configManager.statuses.healthStatus.isGood AND (parts.model5.parts.configManager.statuses.healthStatus.isGood AND (parts.model6.parts.configManager.statuses.healthStatus.isGood AND (parts.model7.parts.configManager.statuses.healthStatus.isGood AND (parts.model8.parts.configManager.statuses.healthStatus.isGood AND parts.model9.parts.configManager.statuses.healthStatus.isGood)))))))),
    hasWarning := parts.model0.parts.configManager.statuses.healthStatus.hasWarning OR (parts.model1.parts.configManager.statuses.healthStatus.hasWarning OR (parts.model2.parts.configManager.statuses.healthStatus.hasWarning OR (parts.model3.parts.configManager.statuses.healthStatus.hasWarning OR (parts.model4.parts.configManager.statuses.healthStatus.hasWarning OR (parts.model5.parts.configManager.statuses.healthStatus.hasWarning OR (parts.model6.parts.configManager.statuses.healthStatus.hasWarning OR (parts.model7.parts.configManager.statuses.healthStatus.hasWarning OR (parts.model8.parts.configManager.statuses.healthStatus.hasWarning OR parts.model9.parts.configManager.statuses.healthStatus.hasWarning)))))))));

          

{attribute 'TcRpcEnable' := '1'}
METHOD _log : BOOL
  VAR_INPUT
    name : STRING;  (* Name of this function block instance *)
  END_VAR
  VAR_IN_OUT
    buffer : LogBuffer;  (* Buffer to write all logging to *)
  END_VAR
  VAR
    subBuffer : LogBuffer;  (* Temporary buffer to write logging by parts (sub-statemachines) to *)
  END_VAR
                  THIS^.parts.model0._log(
    name := 'model0',
    buffer := subBuffer);
THIS^.parts.model1._log(
    name := 'model1',
    buffer := subBuffer);
THIS^.parts.model2._log(
    name := 'model2',
    buffer := subBuffer);
THIS^.parts.model3._log(
    name := 'model3',
    buffer := subBuffer);
THIS^.parts.model4._log(
    name := 'model4',
    buffer := subBuffer);
THIS^.parts.model5._log(
    name := 'model5',
    buffer := subBuffer);
THIS^.parts.model6._log(
    name := 'model6',
    buffer := subBuffer);
THIS^.parts.model7._log(
    name := 'model7',
    buffer := subBuffer);
THIS^.parts.model8._log(
    name := 'model8',
    buffer := subBuffer);
THIS^.parts.model9._log(
    name := 'model9',
    buffer := subBuffer);
LOGGER(
    name := name,
    actualStatus := THIS^.actualStatus,
    previousStatus := THIS^.previousStatus,
    buffer := buffer,
    subBuffer := subBuffer,
    pHealthStatus := ADR(THIS^.statuses.healthStatus),
    pBusyStatus := ADR(THIS^.statuses.busyStatus));

                
END_METHOD
END_FUNCTION_BLOCK

FUNCTION_BLOCK SM_AxesIO
  VAR_INPUT
    {attribute 'OPC.UA.DA' := '1'}
    {attribute 'OPC.UA.DA.Access' := '1'}
    isEnabled : BOOL;  (* Is control enabled? *)
  END_VAR
  VAR_OUTPUT
    {attribute 'OPC.UA.DA' := '1'}
    {attribute 'OPC.UA.DA.Access' := '1'}
    actualStatus : STRING;  (* Current status description *)
    previousStatus : STRING;  (* Previous status description *)
    statuses : AxesIOStatuses;  (* Statuses of the state machine *)
    parts : AxesIOParts;  (* Parts of the state machine *)
  END_VAR

            parts.aziDrive( isEnabled := isEnabled );
parts.ablDrive( isEnabled := isEnabled );
parts.eleDrive( isEnabled := isEnabled );
parts.TA_AZID(
    id := 'TA:AZID',
    typeId := 'AX5206');
parts.TA_ABLD(
    id := 'TA:ABLD',
    typeId := 'AX5206');
parts.TA_ELED(
    id := 'TA:ELED',
    typeId := 'AX5206');
parts.TE_COU(
    id := 'TE:COU',
    typeId := 'EK1100');
parts.TE_EN1(
    id := 'TE:EN1',
    typeId := 'EL5101');
parts.TE_EN2(
    id := 'TE:EN2',
    typeId := 'EL5101');
parts.TE_EN3(
    id := 'TE:EN3',
    typeId := 'EL5101');
parts.TE_EN4(
    id := 'TE:EN4',
    typeId := 'EL5101');
parts.TE_EN5(
    id := 'TE:EN5',
    typeId := 'EL5101');
parts.TE_EN6(
    id := 'TE:EN6',
    typeId := 'EL5101');
parts.TE_EN7(
    id := 'TE:EN7',
    typeId := 'EL5002');
statuses.healthStatus( isGood := parts.aziDrive.statuses.healthStatus.isGood AND (parts.ablDrive.statuses.healthStatus.isGood AND (parts.eleDrive.statuses.healthStatus.isGood AND (parts.TA_AZID.statuses.healthStatus.isGood AND (parts.TA_ABLD.statuses.healthStatus.isGood AND (parts.TA_ELED.statuses.healthStatus.isGood AND (parts.TE_COU.statuses.healthStatus.isGood AND (parts.TE_EN1.statuses.healthStatus.isGood AND (parts.TE_EN1.statuses.healthStatus.isGood AND (parts.TE_EN2.statuses.healthStatus.isGood AND (parts.TE_EN3.statuses.healthStatus.isGood AND (parts.TE_EN4.statuses.healthStatus.isGood AND (parts.TE_EN5.statuses.healthStatus.isGood AND (parts.TE_EN6.statuses.healthStatus.isGood AND parts.TE_EN7.statuses.healthStatus.isGood))))))))))))) );

          

{attribute 'TcRpcEnable' := '1'}
METHOD _log : BOOL
  VAR_INPUT
    name : STRING;  (* Name of this function block instance *)
  END_VAR
  VAR_IN_OUT
    buffer : LogBuffer;  (* Buffer to write all logging to *)
  END_VAR
  VAR
    subBuffer : LogBuffer;  (* Temporary buffer to write logging by parts (sub-statemachines) to *)
  END_VAR
                  THIS^.parts.aziDrive._log(
    name := 'aziDrive',
    buffer := subBuffer);
THIS^.parts.ablDrive._log(
    name := 'ablDrive',
    buffer := subBuffer);
THIS^.parts.eleDrive._log(
    name := 'eleDrive',
    buffer := subBuffer);
THIS^.parts.TA_AZID._log(
    name := 'TA_AZID',
    buffer := subBuffer);
THIS^.parts.TA_ABLD._log(
    name := 'TA_ABLD',
    buffer := subBuffer);
THIS^.parts.TA_ELED._log(
    name := 'TA_ELED',
    buffer := subBuffer);
THIS^.parts.TE_COU._log(
    name := 'TE_COU',
    buffer := subBuffer);
THIS^.parts.TE_EN1._log(
    name := 'TE_EN1',
    buffer := subBuffer);
THIS^.parts.TE_EN2._log(
    name := 'TE_EN2',
    buffer := subBuffer);
THIS^.parts.TE_EN3._log(
    name := 'TE_EN3',
    buffer := subBuffer);
THIS^.parts.TE_EN4._log(
    name := 'TE_EN4',
    buffer := subBuffer);
THIS^.parts.TE_EN5._log(
    name := 'TE_EN5',
    buffer := subBuffer);
THIS^.parts.TE_EN6._log(
    name := 'TE_EN6',
    buffer := subBuffer);
THIS^.parts.TE_EN7._log(
    name := 'TE_EN7',
    buffer := subBuffer);
LOGGER(
    name := name,
    actualStatus := THIS^.actualStatus,
    previousStatus := THIS^.previousStatus,
    buffer := buffer,
    subBuffer := subBuffer,
    pHealthStatus := ADR(THIS^.statuses.healthStatus));

                
END_METHOD
END_FUNCTION_BLOCK

FUNCTION_BLOCK AxesSetTargetProcess EXTENDS BaseProcess
  VAR_INPUT
    {attribute 'OPC.UA.DA' := '1'}
    set : AxesSetTargetProcessArgs;  (* Arguments to be set, before writing do_request TRUE *)
  END_VAR
  VAR_OUTPUT
    {attribute 'OPC.UA.DA' := '1'}
    {attribute 'OPC.UA.DA.Access' := '1'}
    get : AxesSetTargetProcessArgs;  (* Arguments in use by the process, if do_request was accepted *)
  END_VAR

            IF do_request THEN
    do_request_result := request(
    alphaUnits := set.alphaUnits,
    alpha := set.alpha,
    deltaUnits := set.deltaUnits,
    delta := set.delta,
    muUnits := set.muUnits,
    muAlpha := set.muAlpha,
    muDelta := set.muDelta,
    parallax := set.parallax,
    radialVelocity := set.radialVelocity,
    epoch := set.epoch);
    do_request := FALSE;
END_IF;
SUPER^();

          

{attribute 'TcRpcEnable' := '1'}
METHOD start
  VAR_INPUT
    alphaUnits : AxesAlphaUnits;  (* The units in which alpha is given *)
    alpha : LREAL;  (* Right ascention, in the units of the alphaUnits argument *)
    deltaUnits : AxesDeltaUnits;  (* The units in which delta is given *)
    delta : LREAL;  (* Declination, in the units of the deltaUnits argument *)
    muUnits : AxesMuUnits;  (* The units in which muAlpha and muDelta are given *)
    muAlpha : LREAL;  (* Right ascention proper motion, the units of muUmits (do not multiply by cos(delta)!) *)
    muDelta : LREAL;  (* Declination proper motion, in radians/year *)
    parallax : LREAL;  (* Object parallax, in arcseconds *)
    radialVelocity : LREAL;  (* Object radial velocity, in km/s *)
    epoch : LREAL := 2000;  (* Epoch, e.g. 2000.0 *)
  END_VAR
                  THIS^.get.alphaUnits := alphaUnits;
THIS^.get.alpha := alpha;
THIS^.get.deltaUnits := deltaUnits;
THIS^.get.delta := delta;
THIS^.get.muUnits := muUnits;
THIS^.get.muAlpha := muAlpha;
THIS^.get.muDelta := muDelta;
THIS^.get.parallax := parallax;
THIS^.get.radialVelocity := radialVelocity;
THIS^.get.epoch := epoch;
THIS^.statuses.busyStatus( isBusy := TRUE );
THIS^.statuses.healthStatus( isGood := TRUE );

                
END_METHOD

{attribute 'TcRpcEnable' := '1'}
METHOD request : RequestResults
  VAR_INPUT
    alphaUnits : AxesAlphaUnits;  (* The units in which alpha is given *)
    alpha : LREAL;  (* Right ascention, in the units of the alphaUnits argument *)
    deltaUnits : AxesDeltaUnits;  (* The units in which delta is given *)
    delta : LREAL;  (* Declination, in the units of the deltaUnits argument *)
    muUnits : AxesMuUnits;  (* The units in which muAlpha and muDelta are given *)
    muAlpha : LREAL;  (* Right ascention proper motion, the units of muUmits (do not multiply by cos(delta)!) *)
    muDelta : LREAL;  (* Declination proper motion, in radians/year *)
    parallax : LREAL;  (* Object parallax, in arcseconds *)
    radialVelocity : LREAL;  (* Object radial velocity, in km/s *)
    epoch : LREAL := 2000;  (* Epoch, e.g. 2000.0 *)
  END_VAR
                  IF THIS^.statuses.enabledStatus.enabled THEN
    THIS^.start(
        alphaUnits := alphaUnits,
        alpha := alpha,
        deltaUnits := deltaUnits,
        delta := delta,
        muUnits := muUnits,
        muAlpha := muAlpha,
        muDelta := muDelta,
        parallax := parallax,
        radialVelocity := radialVelocity,
        epoch := epoch);
    request := RequestResults.ACCEPTED;
ELSE
    request := RequestResults.REJECTED;
END_IF;

                
END_METHOD
END_FUNCTION_BLOCK

FUNCTION_BLOCK AxesPointProcess EXTENDS BaseProcess
  VAR_INPUT
    state : INT;  (* State of the process *)
    {attribute 'OPC.UA.DA' := '1'}
    set : AxesPointProcessArgs;  (* Arguments to be set, before writing do_request TRUE *)
  END_VAR
  VAR_OUTPUT
    {attribute 'OPC.UA.DA' := '1'}
    {attribute 'OPC.UA.DA.Access' := '1'}
    get : AxesPointProcessArgs;  (* Arguments in use by the process, if do_request was accepted *)
  END_VAR

            IF do_request THEN
    do_request_result := request(
    alphaUnits := set.alphaUnits,
    alpha := set.alpha,
    deltaUnits := set.deltaUnits,
    delta := set.delta,
    muUnits := set.muUnits,
    muAlpha := set.muAlpha,
    muDelta := set.muDelta,
    parallax := set.parallax,
    radialVelocity := set.radialVelocity,
    epoch := set.epoch,
    tracking := set.tracking,
    rotUnits := set.rotUnits,
    rotOffset := set.rotOffset,
    rocOffset := set.rocOffset,
    ronOffset := set.ronOffset,
    doRotOffset := set.doRotOffset,
    doRocOffset := set.doRocOffset,
    doRonOffset := set.doRonOffset);
    do_request := FALSE;
END_IF;
SUPER^();

          

{attribute 'TcRpcEnable' := '1'}
METHOD start
  VAR_INPUT
    alphaUnits : AxesAlphaUnits;  (* The units in which alpha is given *)
    alpha : LREAL;  (* Right ascention, in the units of the alphaUnits argument *)
    deltaUnits : AxesDeltaUnits;  (* The units in which delta is given *)
    delta : LREAL;  (* Declination, in the units of the deltaUnits argument *)
    muUnits : AxesMuUnits;  (* The units in which muAlpha and muDelta are given *)
    muAlpha : LREAL;  (* Right ascention proper motion, the units of muUmits (do not multiply by cos(delta)!) *)
    muDelta : LREAL;  (* Declination proper motion, in radians/year *)
    parallax : LREAL;  (* Object parallax, in arcseconds *)
    radialVelocity : LREAL;  (* Object radial velocity, in km/s *)
    epoch : LREAL := 2000;  (* Epoch, e.g. 2000.0 *)
    tracking : BOOL := TRUE;  (* True to start tracking the object, false to Only do a pointing *)
    rotUnits : AxesMoveUnits;  (* Units of the 'rot', 'roc' and 'ron' arguments (RADIANS, DEGREES, ARCSECONDS, ...) *)
    rotOffset : LREAL;  (* Offset to move the currently active rotator (incompatible with 'roc' and 'ron' args) *)
    rocOffset : LREAL;  (* Offset to move the cassegrain rotation axis (incompatible with 'rot' arg) *)
    ronOffset : LREAL;  (* Offset to move the nasmyth rotation axis (incompatible with 'rot' arg) *)
    doRotOffset : BOOL;  (* True to move the currently active rotator, false to leave it untouched *)
    doRocOffset : BOOL;  (* True to move the cassegrain rotation axis, false to leave it untouched *)
    doRonOffset : BOOL;  (* True to move the nasmyth rotation axis, false to leave it untouched *)
  END_VAR
                  THIS^.get.alphaUnits := alphaUnits;
THIS^.get.alpha := alpha;
THIS^.get.deltaUnits := deltaUnits;
THIS^.get.delta := delta;
THIS^.get.muUnits := muUnits;
THIS^.get.muAlpha := muAlpha;
THIS^.get.muDelta := muDelta;
THIS^.get.parallax := parallax;
THIS^.get.radialVelocity := radialVelocity;
THIS^.get.epoch := epoch;
THIS^.get.tracking := tracking;
THIS^.get.rotUnits := rotUnits;
THIS^.get.rotOffset := rotOffset;
THIS^.get.rocOffset := rocOffset;
THIS^.get.ronOffset := ronOffset;
THIS^.get.doRotOffset := doRotOffset;
THIS^.get.doRocOffset := doRocOffset;
THIS^.get.doRonOffset := doRonOffset;
THIS^.statuses.busyStatus( isBusy := TRUE );
THIS^.statuses.healthStatus( isGood := TRUE );

                
END_METHOD

